		STATE_OPEN: 	(* Waiting for incomming connection *)
				m_SizeSockadr:=SIZEOF(m_AddressInfo);
				m_Socket:= SysSockAccept( m_ServerSocket, ADR(m_AddressInfo), ADR(m_SizeSockadr));
				diError:=State_open;
				IF m_Socket <> SOCKET_INVALID THEN
					xClientConnected:=TRUE;
					(*Set Push-Bit:new V1.5*)
					IF ADR(%MW0)=16#30000000  OR ADR(%MW0)=16#20000000 THEN (*841 or 881*)
						SysSockSetOption(
							diSocket:=m_Socket,
							diLevel:=6,
							diOption:=SOCKET_TCP_NODELAY,
							pOptionValue:=ADR(diOption),
							diOptionLength:=SIZEOF(diOption));
					ELSE
							;
					END_IF
					SysSockIoctl( m_Socket, SOCKET_FIONBIO, ADR(m_NoneBlocking));
					m_State:= STATE_RX;
					diError:=0;
				END_IF

		STATE_RX:
					m_BytesReceived:= SysSockRecv( m_Socket, ADR(m_ReceiveBuffer), SIZEOF(m_ReceiveBuffer), 0);
					CASE m_BytesReceived OF
					-1:(*no data available or error occured*)
						m_ConnectionWatchdog(IN:=TRUE , PT:=tServerTimeOut );
						IF m_connectionWatchdog.Q THEN
							m_State:= STATE_CLOSE;
							m_ConnectionWatchdog(IN:=FALSE);(*reset connection watchdog*)
							diError := 16#8009;
						END_IF
					0:(* socket was "gracefully closed"  *)
						m_State:= STATE_CLOSE;
						diError := 16#8003;
					ELSE
						(* Copy received data into receive buffer *)
						(********************************)
						FOR i:= 0 TO DINT_TO_INT(m_BytesReceived	)-1 DO
							aReceiveBuffer[diReceiveCount]:= m_ReceiveBuffer[i];
							diReceiveCount:=(diReceiveCount+1) MOD SIZEOF(aReceiveBuffer);
						END_FOR

						m_ConnectionWatchdog(IN:=FALSE);(*reset connection watchdog*)
					END_CASE

				(*send data*)
				IF xStartSend	 THEN
					m_State := STATE_TX;
				END_IF

	STATE_TX:	 (* send TCP-message *)
		m_diReturn := SysSockSend(diSocket := m_Socket,
								  pbyBuffer := ADR(ptSendData^[m_count]),(*geändert V1.4 bisher: [0] *)
								  diBufferSize := diSendCount-m_count,
								  diFlags :=m_Flags);
		CASE m_diReturn OF
		-1:	(* ERROR or data could not yet be send (V1.3 due to new FW11) *)
			m_ConnectionWatchdog(IN:=TRUE , PT:=tServerTimeOut );
			IF m_connectionWatchdog.Q THEN
				m_State:= STATE_CLOSE;
				m_ConnectionWatchdog(IN:=FALSE);(*reset connection watchdog*)
				diError := 16#8007;
			END_IF
		0: (* socket was "gracefully closed"  *)
			m_State := STATE_CLOSE;
			diError := 16#8003;
		ELSE (* succesful *)
			m_count:=m_count+m_diReturn;
			IF m_count>=diSendCount THEN
				diError := 16#0000;
				m_State := STATE_RX;
				m_count:=0;
				xStartSend:=FALSE;
			END_IF
			m_ConnectionWatchdog(IN:=FALSE);(*reset connection watchdog*)
		END_CASE


		STATE_CLOSE:	(* Close the server *)

		IF ADR(%MW0)=16#30000000  OR ADR(%MW0)=16#20000000 THEN (*841 or 881*)
			;
		ELSE
			IF m_Socket>=0 THEN
				SysSockShutdown(m_Socket, 0);;(*870*)
			END_IF
		END_IF
		IF m_Socket>=0 THEN
			SysSockClose( m_Socket);
		END_IF
		xClientConnected:= FALSE;
		m_State:= STATE_OPEN; (* Try to open the server again *)
		m_ConnectionWatchdog(IN:=FALSE);(*reset connection watchdog*)

		STATE_ERROR_TRAP: (* Error Read/Write socket  *)
			m_State:= STATE_ERROR_TRAP;

	ELSE  (* Bad FSM code trap  *)
			m_State:= STATE_ERROR_TRAP;
			diError:= 16#8008;
	END_CASE;
ELSE
	IF m_State <> STATE_INIT THEN
		IF ADR(%MW0)=16#30000000  OR ADR(%MW0)=16#20000000 THEN (*841 or 881*)
			;
		ELSE
			IF m_Socket>=0 THEN
				SysSockShutdown(m_Socket, 0);;(*870*)
			END_IF
		END_IF
		IF m_Socket>=0 THEN
			SysSockClose( m_Socket);
		END_IF
		IF ADR(%MW0)=16#30000000  OR ADR(%MW0)=16#20000000 THEN (*841 or 881*)
			;
		ELSE
			IF m_ServerSocket>=0 THEN
				SysSockShutdown(m_ServerSocket, 0);;(*870*)
			END_IF
		END_IF
		IF m_ServerSocket>=0 THEN
			SysSockClose( m_ServerSocket);
		END_IF
		xClientConnected:= FALSE;
		diError:= 0;
		m_State:= STATE_init; (* Try to open the server again *)
		m_ConnectionWatchdog(IN:=FALSE);(*reset connection watchdog*)
	END_IF
END_IF
END_FUNCTION_BLOCK

(* POU Utils Functions/HEXTORAW, ST *)
FUNCTION HEXTORAW : WORD
VAR_INPUT
	pString		: POINTER TO BYTE;
	StringLen	: WORD;
	pData		: POINTER TO BYTE;
END_VAR
VAR
	xl: WORD;
	xi: WORD;
	xr: BYTE;
END_VAR
xl:=0;
xi:=0;

WHILE xi<StringLen DO

	IF pString^>=97 AND pString^<=102 THEN
		xr := pString^ - 87;
	ELSIF pString^>=65 AND pString^<=70 THEN
		xr := pString^ - 55;
	ELSIF pString^>=48 AND pString^<=57 THEN
		xr := pString^ - 48;
	ELSE
		xr := 16;
	END_IF

	IF xr<16 THEN
		IF (xi AND 1)=0 THEN
			pData^ := xr * 16;
		ELSE
			pData^ := pData^ + xr;
			pData := pData + 1;
			xl := xl + 1;
		END_IF
	END_IF

	xi := xi + 1;
	pString := pString + 1;

END_WHILE

HEXTORAW:=xl;
END_FUNCTION

(* POU Utils Functions/RAWTOHEX, ST *)
FUNCTION RAWTOHEX : WORD
VAR_INPUT
	pData: POINTER TO BYTE;
	DataLen: WORD;
	pString: POINTER TO BYTE;
END_VAR
VAR
	xl: WORD;
END_VAR
xl:=0;

WHILE DataLen>0 DO

	pString^ := (pData^ / 16#10) + 48 + (((pData^ / 16#10)/10)*7);
	pString:=pString+1;
	pString^ := (pData^ AND 16#0F)  + 48 + (((pData^ AND 16#0F)/10)*7);
	pString:=pString+1;
	pData:=pData+1;
	DataLen:=DataLen-1;
	xl:=xl+2;

END_WHILE

(*pString^:=0;*)

RAWTOHEX:=xl;
END_FUNCTION

(* POU Utils Functions/SetDataTime, ST *)
FUNCTION SetDataTime : DT
VAR_INPUT
	year : INT;
	month : INT;
	day : INT;
	hour : INT;
	minute : INT;
	second : INT;
END_VAR

VAR
	count : INT;
END_VAR
(* Creazione variabiletipo DT per creare Orario da dare al PLC *)


IF month > 2 THEN
	count := (month - 1) * 30;
	IF month > 7 THEN count := count + SHR(month - 3,1); ELSE count := count + SHR(month - 4,1); END_IF;
	(* chech for leap year and add one day if true *)
	IF SHL(year,14) = 0 THEN count := count + 1; END_IF;
ELSE
	count := (month - 1) * 31;
END_IF;


SetDataTime := DWORD_TO_DT(DATE_TO_DWORD( DWORD_TO_DATE((INT_TO_DWORD(count + day - 1) + SHR(INT_TO_DWORD(year) * 1461 - 2878169, 2)) * 86400))
				+ INT_TO_DWORD(SECOND)
				+ INT_TO_DWORD(MINUTE) * 60
				+ INT_TO_DWORD(HOUR) * 3600);
END_FUNCTION

(* POU Utils/USRLED_Update, ST *)
PROGRAM USRLED_Update
VAR
	OldStatus: en_SYS_Status;

	aFS : ARRAY [0..24] OF FLASHING_SEQUENCE :=
		(Colour:=GREEN,  Frequency:=1,   Relation:=128, Duration:=t#0s,    NextIndex:=0),  (* 0 => RUNNING *)
		(Colour:=ORANGE, Frequency:=1,   Relation:=128, Duration:=t#0s,    NextIndex:=1),  (* 1 => INIT *)
		(Colour:=RED,    Frequency:=4,   Relation:=128, Duration:=t#0s,    NextIndex:=2),  (* 2 => ERROR *)
		(Colour:=RED,    Frequency:=10,  Relation:=128, Duration:=t#0s,    NextIndex:=3),  (* 3 => ALARM *)
		(Colour:=ORANGE, Frequency:=200, Relation:=16,  Duration:=t#100ms, NextIndex:=11), (* 10 *)
		(Colour:=ORANGE, Frequency:=200, Relation:=32,  Duration:=t#100ms, NextIndex:=12),
		(Colour:=ORANGE, Frequency:=200, Relation:=64,  Duration:=t#100ms, NextIndex:=13),
		(Colour:=ORANGE, Frequency:=200, Relation:=128, Duration:=t#100ms, NextIndex:=14),
		(Colour:=ORANGE, Frequency:=200, Relation:=192, Duration:=t#100ms, NextIndex:=15),
		(Colour:=ORANGE, Frequency:=200, Relation:=128, Duration:=t#100ms, NextIndex:=16),
		(Colour:=ORANGE, Frequency:=200, Relation:=64,  Duration:=t#100ms, NextIndex:=17),
		(Colour:=ORANGE, Frequency:=200, Relation:=32,  Duration:=t#100ms, NextIndex:=18),
		(Colour:=ORANGE, Frequency:=200, Relation:=16,  Duration:=t#100ms, NextIndex:=19),
		(Colour:=ORANGE, Frequency:=200, Relation:=8,   Duration:=t#100ms, NextIndex:=10),
		(Colour:=GREEN,  Frequency:=200, Relation:=16,  Duration:=t#100ms, NextIndex:=21), (* 20 *)
		(Colour:=GREEN,  Frequency:=200, Relation:=32,  Duration:=t#100ms, NextIndex:=22),
		(Colour:=GREEN,  Frequency:=200, Relation:=64,  Duration:=t#100ms, NextIndex:=23),
		(Colour:=GREEN,  Frequency:=200, Relation:=128, Duration:=t#100ms, NextIndex:=24),
		(Colour:=GREEN,  Frequency:=200, Relation:=192, Duration:=t#100ms, NextIndex:=25),
		(Colour:=GREEN,  Frequency:=200, Relation:=128, Duration:=t#100ms, NextIndex:=26),
		(Colour:=GREEN,  Frequency:=200, Relation:=64,  Duration:=t#100ms, NextIndex:=27),
		(Colour:=GREEN,  Frequency:=200, Relation:=32,  Duration:=t#100ms, NextIndex:=28),
		(Colour:=GREEN,  Frequency:=200, Relation:=16,  Duration:=t#100ms, NextIndex:=29),
		(Colour:=GREEN,  Frequency:=200, Relation:=8,   Duration:=t#100ms, NextIndex:=20);

	pFS : POINTER TO FLASHING_SEQUENCE;


END_VAR
IF Sys.Status <> OldStatus THEN

	OldStatus:=Sys.Status;

	CASE OldStatus OF

		S_STARTUP:
			pFS:=ADR(aFS);
			SET_FLASHING_SEQUENCE(EN:=TRUE, POINTER_TO_POINTER_TO_ARRAY:=ADR(pFS));
			SET_FLASHING_SEQUENCE_INDEX(EN:=TRUE, IMMEDIATE:=FALSE, INDEX:=1);
			START_FLASHING_SEQUENCE(EN:=TRUE);

		S_RUNNING:
			SET_FLASHING_SEQUENCE_INDEX(EN:=TRUE, IMMEDIATE:=TRUE, INDEX:=0);

	END_CASE

END_IF
END_PROGRAM

(* POU ConteggioGAS1, ST *)
PROGRAM ConteggioGAS1

VAR RETAIN
	Conteggio_GAS1: DINT;
END_VAR
(* Attenzione Portata GAS Caldaia n.3 SEVESO *)


Conteggio_GAS1:=Conteggio_GAS1+1;
END_PROGRAM
ACTION Offset:
(* Offset *)

IF ChangeGAS1 THEN
	Conteggio_GAS1:=OffsetGAS1;
	ChangeGAS1:=FALSE;
END_IF
END_ACTION

(* POU ConteggioGAS2, ST *)
PROGRAM ConteggioGAS2

VAR RETAIN
	Conteggio_GAS2: DINT;
END_VAR
(* Attenzione Portata GAS per Caldaia CAL02 e CAL03 *)

Conteggio_GAS2:=Conteggio_GAS2+1;
END_PROGRAM
ACTION Offset:
(* Offset *)

IF ChangeGAS2 THEN
	Conteggio_GAS2:=OffsetGAS2;
	ChangeGAS2:=FALSE;
END_IF
END_ACTION

(* POU Plant/SYS_Proc, ST *)
PROGRAM SYS_Proc
VAR
(*	fALARM_PB		:FLT_TAP;
	fALARM_TB		:FLT_TAP;
	fALARM_PM		:FLT_TAP; *)

(*	fGZB_ST			:FLT_TAP;  (* GATEWAY ZIGBEE *)*)
(*	fVPN_ST1		:FLT_TAP;  (* VPN CONNECT *)*)
	fVPN_ST2		:FLT_TAP;  (* VPN STATUS *)
(*	fKEY_CT_ST		:FLT_TAP;  (* DOOR1 *)*)
(*	fKEY_SCT_ST		:FLT_TAP;  (* DOOR2 *)*)
	fKEY_QE_ST		:FLT_TAP;  (* DOOR3 *)

END_VAR
(*************** ISPESL *****************)
(*
fALARM_PB(IN:=ALARM_PB);
IF fALARM_PB.EVH THEN
	LogEv(EL_AlarmStop,EO_PBV,1,1,'Over_Pressure_Alarm');
END_IF

fALARM_TB(IN:=ALARM_TB);
IF fALARM_TB.EVH THEN
	LogEv(EL_AlarmStop,EO_TBV,1,1,'Over_Temperature_Alarm');
END_IF

fALARM_PM(IN:=ALARM_PM);
IF fALARM_PM.EVH THEN
	LogEv(EL_AlarmStop,EO_PMV,1,1,'Under_Pressure_Alarm');
END_IF
*)
(****************************************)

(*### VPN Connection Check ###*)(*
fVPN_ST1(IN:=VPN_ST1);
IF fVPN_ST1.EVH THEN
	LogEv(EL_Log,EO_VPN,1,1,'CONNECT_ON');
END_IF
IF fVPN_ST1.EVL THEN
	LogEv(EL_Log,EO_VPN,1,2,'CONNECT_OFF');
END_IF*)

(*### VPN Status Check ###*)
fVPN_ST2(IN:=VPN_ST2);
IF fVPN_ST2.EVH THEN
	LogEv(EL_Log,EO_VPN,1,3,'STATUS_UP');
END_IF
IF fVPN_ST2.EVL THEN
	LogEv(EL_Wrn,EO_VPN,1,4,'STATUS_DOWN');
END_IF

(*### DOOR01 Status Check ###*)(*
fKEY_CT_ST(IN:=KEY_CT_ST);
IF fKEY_CT_ST.EVH THEN
	LogEv(EL_Log,EO_DOOR,1,2,'Centrale_termica_Close');
END_IF
IF fKEY_CT_ST.EVL THEN
	LogEv(EL_Wrn,EO_DOOR,1,1,'Centrale_termica_Open');
END_IF*)

(*### DOOR02 Status Check ###*)(*
fKEY_SCT_ST(IN:=KEY_SCT_ST);
IF fKEY_SCT_ST.EVH THEN
	LogEv(EL_Log,EO_DOOR,2,2,'Sottocentrale_termica_Close');
END_IF
IF fKEY_SCT_ST.EVL THEN
	LogEv(EL_Wrn,EO_DOOR,2,1,'Sottocentrale_termica_Open');
END_IF*)

(*### DOOR03 Status Check ###*)
fKEY_QE_ST(IN:=KEY_QE_ST);
IF fKEY_QE_ST.EVH THEN
	LogEv(EL_Log,EO_DOOR,3,2,'Quadro_Close');
END_IF
IF fKEY_QE_ST.EVL THEN
	LogEv(EL_Wrn,EO_DOOR,3,1,'Quadro_Open');
END_IF
END_PROGRAM

(* POU Utils Functions/AVERAGE_DINT, ST *)
FUNCTION_BLOCK AVERAGE_DINT
VAR_INPUT
	IN: 	DINT;
END_VAR
VAR_OUTPUT
	HI:		DINT;
	AVG:	DINT;
	LOW:	DINT;
	ERR:	BOOL;
END_VAR
VAR
	sum:	REAL;
	cnt:	WORD;
END_VAR
IF cnt>=65000 THEN
	ERR:=TRUE;
	Read();
	sum := sum - DINT_TO_REAL(AVG);
	cnt := cnt - 1;
END_IF

sum := sum + DINT_TO_REAL(IN);
cnt := cnt + 1;

IF IN<LOW THEN LOW:=IN; END_IF
IF IN>HI  THEN HI :=IN; END_IF
END_FUNCTION_BLOCK
ACTION Read:
AVG := REAL_TO_DINT(sum/cnt);
END_ACTION
ACTION Reset:
HI:=IN;
AVG:=IN;
LOW:=IN;
ERR:=FALSE;

sum:=DINT_TO_REAL(IN);
cnt:=1;
END_ACTION

(* POU Utils Functions/AVERAGE_INT, ST *)
FUNCTION_BLOCK AVERAGE_INT
VAR_INPUT
	IN: 	INT;
END_VAR
VAR_OUTPUT
	HI:		INT;
	AVG:	INT;
	LOW:	INT;
	ERR:	BOOL;
END_VAR
VAR
	sum:	DINT;
	cnt:	WORD;
END_VAR
IF cnt>=65000 THEN
	ERR:=TRUE;
	Read();
	sum := sum - AVG;
	cnt := cnt - 1;
END_IF

sum := sum + IN;
cnt := cnt + 1;

IF IN<LOW THEN LOW:=IN; END_IF
IF IN>HI  THEN HI :=IN; END_IF
END_FUNCTION_BLOCK
ACTION Read:
AVG := DINT_TO_INT(sum/cnt);
END_ACTION
ACTION Reset:
HI:=IN;
AVG:=IN;
LOW:=IN;
ERR:=FALSE;

sum:=IN;
cnt:=1;
END_ACTION

(* POU Utils Functions/AVERAGE_T, ST *)
FUNCTION_BLOCK AVERAGE_T
VAR_INPUT
	IN: 	INT;
END_VAR
VAR_OUTPUT
	HI:		INT;
	AVG:	INT;
	LOW:	INT;
	ERR:	BOOL;
END_VAR
VAR
	sum:	DINT;
	cnt:	WORD;
END_VAR
IF cnt>=65000 THEN
	ERR:=TRUE;
	Read();
	sum := sum - AVG;
	cnt := cnt + 1;
END_IF

sum := sum + IN;
cnt := cnt + 1;

IF IN<LOW THEN  LOW:=IN; END_IF
IF IN>HI  THEN HI :=IN; END_IF
END_FUNCTION_BLOCK
ACTION Read:
AVG := DINT_TO_INT(sum/cnt);
END_ACTION
ACTION Reset:
HI:=IN;
AVG:=IN;
LOW:=IN;
ERR:=FALSE;

sum:=IN;
cnt:=1;
END_ACTION

(* POU Utils Functions/COPY_32SWAP16, ST *)
FUNCTION COPY_32SWAP16:BOOL
VAR_INPUT
	pSourceAddress		:POINTER TO ARRAY[1..2] OF WORD;
	pDestinationAddress	:POINTER TO ARRAY[1..2] OF WORD;
END_VAR
VAR
END_VAR
pDestinationAddress^[1]:=pSourceAddress^[2];
pDestinationAddress^[2]:=pSourceAddress^[1];
END_FUNCTION

(* POU Utils/CSV_Log, ST *)
FUNCTION CSV_Log : BOOL
VAR_INPUT
END_VAR
VAR CONSTANT
	LogFileName:STRING:='S:\LOGS_ID3V3.CSV';
END_VAR
VAR
	s1 : STRING(180);
	hFile: 	DWORD;
END_VAR
(* Check file presence *)
hFile:=SysFileOpen(LogFileName,'r');
IF hFile=0 THEN
	(*** File not exist *** Create file and write header *)
	hFile:=SysFileOpen(LogFileName,'w');
	IF hFile<>0 THEN
		(* Write CSV header *)
		s1:='DATE-TIME;T-SA;T-S02;T-S03;T-S04;T-S05;T-S06;T-S07;';
		SysFileWrite(hFile, ADR(s1), LEN(s1));
		s1:='PORT01-Flow;PORT01-Cnt;GAS01-Cnt;GAS02-Cnt;';
		SysFileWrite(hFile, ADR(s1), LEN(s1));
		s1:='CTB250-Power;CTB250-KWH;CTB250-GWH';
		SysFileWrite(hFile, ADR(s1), LEN(s1));
		SysFileWrite(hFile, ADR(Logger_CRLF), LEN(Logger_CRLF));
	END_IF
ELSE
	(*** File exist *** Close file and reopen in append mode *)
	SysFileClose(hFile);
	hFile:=SysFileOpen(LogFileName,'a');
END_IF

(* Log to file *)
IF hFile<>0 THEN
	(* Date stamp *)
	s1:=REPLACE( Sys.Time_LogString , ' ' , 1 , 11 );
	SysFileWrite(hFile, ADR(s1), LEN(s1));
	(* Log data *)
	s1:=CONCAT(';', INT_TO_STRING(TT_S01) );
	s1:=CONCAT(s1 , ';' );
	s1:=CONCAT(s1 , INT_TO_STRING(TPV02.ValoreScalato) );
	s1:=CONCAT(s1 , ';' );
	s1:=CONCAT(s1 , INT_TO_STRING(TPV03.ValoreScalato) );
	s1:=CONCAT(s1 , ';' );
	s1:=CONCAT(s1 , INT_TO_STRING(TPV04.ValoreScalato) );
	s1:=CONCAT(s1 , ';' );
	s1:=CONCAT(s1 , INT_TO_STRING(TPV05.ValoreScalato) );
	s1:=CONCAT(s1 , ';' );
	s1:=CONCAT(s1 , INT_TO_STRING(TPV06.ValoreScalato) );
	s1:=CONCAT(s1 , ';' );
	s1:=CONCAT(s1 , INT_TO_STRING(TPV07.ValoreScalato) );
	SysFileWrite(hFile, ADR(s1), LEN(s1));
	s1:=CONCAT(';', DINT_TO_STRING(PORT01.ValoreScalato/1000) );
	s1:=CONCAT(s1 , ';' );
	s1:=CONCAT(s1 , DINT_TO_STRING(PortataTotalePORT01) );
	s1:=CONCAT(s1 , ';' );
	s1:=CONCAT(s1 , DINT_TO_STRING(ConteggioGAS1.Conteggio_GAS1) );
	s1:=CONCAT(s1 , ';' );
	s1:=CONCAT(s1 , DINT_TO_STRING(ConteggioGAS2.Conteggio_GAS2) );
(*	s1:=CONCAT(s1 , DINT_TO_STRING(PortataTotaleGAS01) );
	s1:=CONCAT(s1 , ';' );
	s1:=CONCAT(s1 , DINT_TO_STRING(PortataTotaleGAS02) );*)
	SysFileWrite(hFile, ADR(s1), LEN(s1));
	s1:=CONCAT(';', DINT_TO_STRING(REAL_TO_DINT(CTB250.POWER_KW)) );
	s1:=CONCAT(s1 , ';' );
	s1:=CONCAT(s1 , DWORD_TO_STRING(CTB250_ENERGY) );
	SysFileWrite(hFile, ADR(s1), LEN(s1));

	(* Add line CRLF and close *)
	SysFileWrite(hFile, ADR(Logger_CRLF), LEN(Logger_CRLF));
	SysFileClose(hFile);
END_IF
END_FUNCTION

(* POU Utils Functions/FLT_EVENT, ST *)
FUNCTION_BLOCK FLT_EVENT
VAR_INPUT
	IN		: BOOL;
	INITEV	: BOOL:=TRUE;
END_VAR
VAR_OUTPUT
	EVH		: BOOL;
	EVL		: BOOL;
END_VAR
VAR
	init	: BOOL:=FALSE;
	old		: BOOL;
END_VAR
EVH:=FALSE;
EVL:=FALSE;

IF NOT init THEN
	init:=TRUE;
	IF INITEV THEN
		old := NOT IN;
	ELSE
		old := IN;
	END_IF
END_IF

IF old<>IN THEN
	old:=IN;
	IF IN THEN EVH:=TRUE; ELSE EVL:=TRUE; END_IF
END_IF
END_FUNCTION_BLOCK

(* POU Utils Functions/FLT_TIME, ST *)
FUNCTION_BLOCK FLT_TIME
VAR_INPUT
	IN		: BOOL;
	TTAP	: TIME:=T#5s;
	INITEV	: BOOL:=TRUE;
END_VAR
VAR_OUTPUT
	OUT		: BOOL;
	EVH		: BOOL;
	EVL		: BOOL;
END_VAR
VAR
	init	: BOOL:=FALSE;
	timer	: TON;
END_VAR
EVH:=FALSE;
EVL:=FALSE;

IF NOT init THEN
	init := TRUE;
	IF INITEV THEN
		OUT  := NOT IN;
	ELSE
		OUT  := IN;
	END_IF
END_IF

IF OUT<>IN THEN
	timer(IN:=TRUE,PT:=TTAP);
	IF timer.Q THEN
		OUT:=IN;
		timer(IN:=FALSE);
		IF OUT THEN EVH:=TRUE; ELSE EVL:=TRUE; END_IF
	END_IF
ELSE
	timer(IN:=FALSE);
END_IF
END_FUNCTION_BLOCK

(* POU Utils Functions/LINEAR, ST *)
FUNCTION LINEAR : REAL (* Linear interpolation *)
VAR_INPUT
	X_In	: REAL;
	P1_X	: REAL;
	P1_Y	: REAL;
	P2_X	: REAL;
	P2_Y	: REAL;
END_VAR
VAR
END_VAR
LINEAR:=P1_Y+(((P2_Y-P1_Y)*(X_In-P1_X))/(P2_X-P1_X));
END_FUNCTION

(* POU Utils Functions/LINEAR_BAD, ST *)
FUNCTION LINEAR_BAD : INT (* Linear interpolation *)
VAR_INPUT
	PuntoMinX	: INT;
	PuntoMaxX	: INT;
	ValIn		: INT;
	PuntoMinY	: REAL;
	PuntoMaxY	: REAL;
	Decimali	: BYTE;
END_VAR
VAR
	Gain				: REAL;
	PuntoMinX_R			: REAL;
	PuntoMaxX_R			: REAL;
	Linearizzazione_R	: REAL;
END_VAR
PuntoMinX_R:=INT_TO_REAL(PuntoMinX);
PuntoMaxX_R:=INT_TO_REAL(PuntoMaxX);

Gain:=(PuntoMaxX_R-PuntoMinX_R)/(PuntoMaxY-PuntoMinY);	(* Calcolo in guadagno per la linarizzazione *)
Linearizzazione_R:=PuntoMinx+(Gain*(ValIn-PuntoMinY));	(* Ottengo il valore linearizzato *)

LINEAR_BAD:=REAL_TO_INT(Linearizzazione_R*(EXPT(10, Decimali)));  (* Ottengo intero con i decimai voluti *)
END_FUNCTION

(* POU TCP_Logger/LogTrig, ST *)
FUNCTION LogTrig : BOOL
VAR
	s1 : STRING(160);
	i  : BYTE;
END_VAR
(*---------------------------------------------------------------*)
	Logger_Head();
(*---------------------------------------------------------------*)

(* Insert TPVs *)
(*
s1:=CONCAT('&TPV=',INT_TO_STRING(TPV01.AVG));
(*TPV01.Mean_Reset(); *)
s1:=CONCAT(s1,';'); s1:=CONCAT(s1,INT_TO_STRING(TPV02.ValoreScalato));
s1:=CONCAT(s1,';'); s1:=CONCAT(s1,INT_TO_STRING(TPV03.ValoreScalato));
s1:=CONCAT(s1,';'); s1:=CONCAT(s1,INT_TO_STRING(TPV04.ValoreScalato));
s1:=CONCAT(s1,';'); s1:=CONCAT(s1,INT_TO_STRING(TPV05.ValoreScalato));
s1:=CONCAT(s1,';'); s1:=CONCAT(s1,INT_TO_STRING(TPV06.ValoreScalato));
s1:=CONCAT(s1,';'); s1:=CONCAT(s1,INT_TO_STRING(TPV07.ValoreScalato));
s1:=CONCAT(s1,';'); s1:=CONCAT(s1,INT_TO_STRING(TPV08.ValoreScalato));
s1:=CONCAT(s1,';'); s1:=CONCAT(s1,INT_TO_STRING(TPV09.ValoreScalato));

ADDSTRING(ADR(Logger.TData), ADR(s1), Logger.TLen);
*)

TPV01.AddLogData();
TPV02.AddLogData();
TPV03.AddLogData();
TPV04.AddLogData();
TPV05.AddLogData();
TPV06.AddLogData();
TPV07.AddLogData();
TPV08.AddLogData();
TPV09.AddLogData();

THER01.AddLogData();
THER02.AddLogData();
THER03.AddLogData();
THER04.AddLogData();

CIRD01.AddLogData();
CIRD02.AddLogData();

EV02.AddLogData();
EV03.AddLogData();

CAL02.AddLogData(CLIM:=CAL02_Clima);
CAL03.AddLogData(CLIM:=CAL03_Clima);

(* Insert contabilizers  *)

s1:=CONCAT('&PORT01=',DINT_TO_STRING(PORT01.ValoreScalato));
s1:=CONCAT(s1,';'); s1:=CONCAT(s1,DINT_TO_STRING(PortataTotalePORT01));
s1:=CONCAT(s1,';'); s1:=CONCAT(s1,BYTE_TO_STRING(PORT01.Status_Log));
ADDSTRING(ADR(Logger.TData), ADR(s1), Logger.TLen);


(*
s1:=CONCAT('&GAS01=',DINT_TO_STRING(PortataTotaleGAS01));
s1:=CONCAT(s1,';'); s1:=CONCAT(s1,BYTE_TO_STRING(GAS01.Status_Log));
ADDSTRING(ADR(Logger.TData), ADR(s1), Logger.TLen);

s1:=CONCAT('&GAS02=',DINT_TO_STRING(PortataTotaleGAS02));
s1:=CONCAT(s1,';'); s1:=CONCAT(s1,BYTE_TO_STRING(GAS02.Status_Log));
ADDSTRING(ADR(Logger.TData), ADR(s1), Logger.TLen);
*)

(* Registro il nuovo conteggio *)


s1:=CONCAT('&GAS01=',DINT_TO_STRING(ConteggioGAS1.Conteggio_GAS1));
s1:=CONCAT(s1,';'); s1:=CONCAT(s1,BYTE_TO_STRING(GAS01.Status_Log));
ADDSTRING(ADR(Logger.TData), ADR(s1), Logger.TLen);

s1:=CONCAT('&GAS02=',DINT_TO_STRING(ConteggioGAS2.Conteggio_GAS2));
s1:=CONCAT(s1,';'); s1:=CONCAT(s1,BYTE_TO_STRING(GAS02.Status_Log));
ADDSTRING(ADR(Logger.TData), ADR(s1), Logger.TLen);


(*CTBSCAN01.AddLogData( MBUS:=MBUS01 ); ==> TOO BIG! *)
CTB250.AddLogData( ENERGY_WH:=CTB250_ENERGY_WH,	ENERGY:=CTB250_ENERGY );

SCA_Proc.AddLogData();

(*---------------------------------------------------------------*)
	Logger_Send();
(*---------------------------------------------------------------*)
END_FUNCTION

(* POU Utils Functions/MEMCLR, ST *)
FUNCTION MEMCLR:BOOL
VAR_INPUT
	pDestinationAddress:POINTER TO ARRAY[1..2] OF BYTE;
	BytesToClear:WORD;
END_VAR
VAR
END_VAR
WHILE (BytesToClear > 0) DO
	pDestinationAddress^[1]:=0;
	pDestinationAddress:=ADR(pDestinationAddress^[2]); (* increment destination *)
	BytesToClear:=BytesToClear -1; (* decrement number of bytes to copy *)
END_WHILE
END_FUNCTION

(* POU Plant_Objects/obj_CAL_01, ST *)
FUNCTION_BLOCK obj_CAL_01
(* === CALDAIA generica con comando digitale, Set point analogico feedback potenza e stato caldaia  ===
   VERSIONE 01 REALIZZATA DA MORENO E TESTA SU IMPIANTO SAN FELICE ID 003 CLV
	Caldaia controllata con: 	- uscita analogica
								- comando on/off. 
								- Reset Blocco Bruciatore
	
	come feedback si sapetta: 	- riferimento analogico per potenza
								- Stato Presenza fiamma per segnalazione Caldaia accesa
								- Stato Blocco Brucitaore
*)
VAR_INPUT

	ID				: BYTE;			(* Impostazione *)
	LimiteMAXSetPoint: INT;			(* Da Settare : limite massimo da assegnare al riferimento analogico onde evitare di mal comndare la caldaia *)
	LimiteMinSetPoint: INT;			(* Da Settare : limite massimo da assegnare al riferimento analogico onde evitare di mal comndare la caldaia *)

	SetPointManuale: INT; 			(* SetPoint forazato in manuale serve per escludere la curva climatica locale *)
	AbilitaSetPointManuale : BOOL ; (* Abilita il funzionamento col set point Manaule Escludendo la curva cliamtica *)

	Run				: BOOL;			(* Controllo/ comando esterno generalmente da Crono *)


(* ingressi fisici analogici *)

	AI_Potenza		:INT;			(* Riferimento della potenza erogata dalla Caldaia *)

(* ingressi fisici digitali *)

	CAL_ST : BOOL;					(* Stato della Caldia Accesa Spenta - Presenza Fiamma *)
	ALARM_CAL:BOOL;					(* Caldaia in BLocco  *)
	PresenzaFiamma:BOOL;			(* Segnalazione Presenza Fiamma *)


	CmdCALAuto_MAN: BOOL;			(* Modalaita di Funzionamento Caldaia : 0 Automatico. 1 Manuale Solitamnete Selettore a bordo Caldaia *)

	TCP_ResetCAL:BOOL;				(* Comando Reset Caldaia da Remoto via FTP *)
	Rearm:BOOL;						(* Comando Reset Caldaia da locale pulsante WebVisu *)

END_VAR
VAR_IN_OUT
	CLIM		  : typ_Clima;
END_VAR
VAR_OUTPUT
	Curve_Temp		: INT;
	AO_SetPoint		:INT;

	CAL_EN			:BOOL;
	DO_RIARMO		:BOOL;

	(* Status *)
	Status_Log	: BYTE;
	Status_Vis 	: DWORD;
END_VAR
VAR
	InitOK		: BOOL;

	Alarm: BOOL;
	Warning:BOOL;
	Warning2: BOOL;

	Curve 		: CHARCURVE;
	Curve_Err 	: BYTE;


	(* Timer manage switch on/off delay *)
	Delay		: 	TONOF;


	Potenza:INT;
	SetPoint:INT;

	fSTATO_CAL: FLT_TAP;
	fALARM_CAL: FLT_TAP;
	fCALAuto_MAN: FLT_TAP;



	TP_RIARMO: TP:=(PT:=t#5s);



	MAXTentativi: BYTE;
	Trig_TP_RIARMO: R_TRIG;




END_VAR

VAR_INPUT RETAIN

	(* Timings *)
	OnDelay		:	TIME;	(* Switch on delay *)
	OffDelay	:	TIME;	(* Switch off delay *)


END_VAR
(* Check initialization *)
(*IF NOT InitOK THEN Init(); END_IF*)

(* Recupero della curva cliamtica *)

IF NOT CLIM.InitOK THEN Clima_Default(); END_IF;
(* Calculate Setpoint *)
Curve(	IN:= T_AMB,	N:= 5, P:= CLIM.Points,
		OUT=> Curve_Temp, ERR=> Curve_Err );
IF Curve_Err>0  THEN
	IF NOT Warning THEN
		Warning:=TRUE;
		LogEv(EL_Wrn,EO_CAL,ID,2,'Climatic_Error');
	END_IF
ELSE
	Warning:=FALSE;
END_IF


(* Scelta del set point della cladaia o vien preso dalla curva cliamtica o da un riferimento esterno *)
IF AbilitaSetPointManuale THEN
	SetPoint:=(SetPointManuale + OffsetSetPointManuale);
ELSE
	SetPoint:=Curve_Temp*10;
END_IF


(* Linearizzazione segnali analogici *)

(* calcolao il valore delset point da passare alla scheda di uscita  analogica *)
SetPoint:=LIMIT(LimiteMinSetPoint,SetPoint,LimiteMAXSetPoint);
AO_SetPoint:=LINEAR_BAD(0, 32767, SetPoint, 0,1500 , 0);

(* trovo Valore della potenza della Caldaia *)
Potenza:=LINEAR_BAD(0, 100, AI_Potenza, 6553, 32767, 0);
Potenza:=LIMIT(0,Potenza,100);




(* Comando fisico alla caldaia Solito Ton e TOFF *)
IF OffDelay<t#1s THEN OffDelay:=t#1s;END_IF;
IF OnDelay<t#1m THEN OffDelay:=t#1m;END_IF;

Delay(IN:=RUN,PT_OF:=OffDelay,PT_ON:=OnDelay + WORD_TO_TIME(1000*ID));    (* Ritardo all'accensione e allo Spegnimento *)

(* Controllo On/Off Caldaia *)
IF Delay.OUT AND (NOT Alarm) AND NOT CmdCALAuto_MAN THEN
	CAL_EN:=TRUE;
 ELSE
	CAL_EN:=FALSE;
END_IF


(** Riarmo Reset Caldaia tolgo tensione per 5 secondi alla caldaia ***)

TP_RIARMO(IN:=Rearm OR TCP_ResetCAL AND ALARM_CAL );
DO_RIARMO:=TP_RIARMO.Q;
Rearm:=FALSE;
TCP_ResetCAL:=FALSE;

Trig_TP_RIARMO(CLK:=TP_RIARMO.Q);
IF Trig_TP_RIARMO.Q THEN MAXTentativi:=MAXTentativi+1;END_IF
IF MAXTentativi >5 THEN
	LogEv(EL_Alarm,EO_CAL,ID,14,'Reset_Caldaia_non_riuscito');
	MAXTentativi:=0;
END_IF

(* Stato CALDAIA *)
fALARM_CAL(IN:=ALARM_CAL);
IF fALARM_CAL.EVH THEN
	LogEv(EL_Alarm,EO_CAL,ID,5,'Caldaia_In_Blocco');
	Alarm:=TRUE;
END_IF
IF fALARM_CAL.EVL THEN
	LogEv(EL_Alarm,EO_CAL,ID,6,'CALDAIA_Sbloccata');
	MAXTentativi:=0;
	Alarm:=FALSE;
END_IF

(* Stato CALDAIA CALDAIA in Mauale  *)
fCALAuto_MAN(IN:=CmdCALAuto_MAN);
IF fCALAuto_MAN.EVH THEN
	LogEv(EL_wrn,EO_CAL,ID,12,'Caldaia_In_Manuale');
	Warning2:=TRUE;
END_IF
IF fCALAuto_MAN.EVL THEN
	LogEv(EL_Log,EO_CAL,ID,13,'CALDAIA_in_Automatico');
	Warning2:=FALSE;
END_IF


(* Stato CALDAIA *)
fSTATO_CAL(IN:=CAL_ST);
IF fSTATO_CAL.EVH THEN
	LogEv(EL_Log,EO_CAL,ID,10,'Caldaia_RUN_Presenza_Fiamma');
	MAXTentativi:=0;
END_IF
IF fSTATO_CAL.EVL THEN
	LogEv(EL_Log,EO_CAL,ID,11,'CALDAIA_STOP_Assenza_Fiamma');
END_IF



(* Seganalzione stato Caldaia *)
  IF Alarm THEN
		Status_Log:=2; Status_Vis:=16#2020F0;
		AO_SetPoint:=0;
	ELSIF Warning OR Warning2 THEN
			Status_Log:=1; Status_Vis:=16#20F0F0;
    ELSE
		Status_Log:=0;
		Status_Vis:=16#006000;
END_IF
END_FUNCTION_BLOCK
ACTION AddLogData:
Logger.s1:=INSERT('&CAL=',BYTE_TO_STRING(ID),4);
IF ID<10 THEN Logger.s1:=INSERT(Logger.s1,'0',4); END_IF

Logger.s1:=CONCAT(Logger.s1,INT_TO_STRING(SetPoint));
Logger.s1:=CONCAT(Logger.s1,';');
Logger.s1:=CONCAT(Logger.s1,SEL(Run,'0','100'));
Logger.s1:=CONCAT(Logger.s1,';');

Logger.s1:=CONCAT(Logger.s1,WORD_TO_STRING(Status_Log));

Logger.s1:=CONCAT(Logger.s1,';');
Logger.s1:=CONCAT(Logger.s1,INT_TO_STRING(OffsetSetPointManuale));			(* non pesente in quanto non c'è lo scambiatore *)
Logger.s1:=CONCAT(Logger.s1,';');
Logger.s1:=CONCAT(Logger.s1,INT_TO_STRING(Potenza)); 						(* Potenza Caldaia *)
Logger.s1:=CONCAT(Logger.s1,';');
Logger.s1:=CONCAT(Logger.s1,INT_TO_STRING(BOOL_TO_INT(PresenzaFiamma))); 				(* Presenza Fiamma *)
Logger.s1:=CONCAT(Logger.s1,';');
Logger.s1:=CONCAT(Logger.s1,INT_TO_STRING(0)); 								(* non recuperabile Temp. Mandata da Caldaia*)
Logger.s1:=CONCAT(Logger.s1,';');
Logger.s1:=CONCAT(Logger.s1,'3');	 											(* Temp. Tipo Caldaia Sempre in questo punto
																				0 = > Albino
																				1 = > Caldaia con Protocollo LON
																				2 = > comandi digitali senza set point 
																				3 = > comandi digitali con set point *)
Logger.s1:=CONCAT(Logger.s1,';');
Logger.s1:=CONCAT(Logger.s1,INT_TO_STRING(BOOL_TO_INT(CmdCALAuto_MAN)));	 					(* 0 caldia in Automatico : 1= Caldaia in Manuale *)



ADDSTRING(ADR(Logger.TData), ADR(Logger.s1), Logger.TLen);
END_ACTION
ACTION Clima_Default:
IF CLIM.Points[0].X=0 THEN
CLIM.Points[0].X:=-100; CLIM.Points[0].Y:=800;
CLIM.Points[1].X:=0 ; CLIM.Points[1].Y:=750;
CLIM.Points[2].X:= 100;  CLIM.Points[2].Y:=700;
CLIM.Points[3].X:= 150; CLIM.Points[3].Y:=650;
CLIM.Points[4].X:= 200; CLIM.Points[4].Y:=400;
END_IF
CLIM.InitOK:=TRUE;
LogEv(EL_Wrn,EO_CAL,ID,1,'Climatic_default');
END_ACTION
ACTION Init:
(* End initialization *)
InitOK:=TRUE;
END_ACTION

(* POU Utils Functions/TONOF, ST *)
FUNCTION_BLOCK TONOF
VAR_INPUT
	IN		: BOOL;
	PT_ON	: TIME; (* time to pass, before OUT is set *)
	PT_OF	: TIME; (* time to pass, before OUT is reset *)
END_VAR
VAR_OUTPUT
	OUT		: BOOL;
END_VAR
VAR
	timer	: TON;
END_VAR
IF IN<>OUT THEN
	timer(IN:=TRUE,PT:=SEL(IN,PT_OF,PT_ON));
	IF timer.Q THEN OUT:=IN; END_IF
ELSE
	timer(IN:=FALSE);
END_IF
END_FUNCTION_BLOCK

(* POU Plant_Objects/obj_CIRD_01, ST *)
FUNCTION_BLOCK obj_CIRD_01
(* === CIRCOLATORE GEMELLARE STANDARD ===
   VERSIONE 01 REALIZZATA DA MORENO E TESTA SU IMPIANTO SAN FELICE ID 003 CLV
*)

VAR_INPUT
	(* Settings *)
	ID				: BYTE;

	(* Forzature da FTP *)
	CIR_RUN_REQ		: BOOL; (* Richiesta di avvio Circolatore  - Vince sullo stato del ciclo *)
	CIR_STOP_REQ	: BOOL; (* Richiesta di Stop Circolatore - Vince sullo stato del ciclo *)

	(* Ingressi Fisici  *)
	PumpA_AL		: BOOL; (* Allarme Pump A - Salvamotore Intervenuto *)
	PumpB_AL		: BOOL; (* Allarme Pump B - Salvamotore Intervenuto *)
	PumpA_ST		: BOOL; (* Stato Pump A - Generalmente Stato del Contattore *)
	PumpB_ST		: BOOL; (* Stato Pump B - Generalmente Stato del Contattore *)
	PumpA_AUTO		: BOOL; (* Pump A in 1=Automatico o 0=Manuale *)
	PumpB_AUTO		: BOOL; (* Pump B in 1=Automatico o 0=Manuale *)

	(* Controls *)
	OnOff			: BOOL;		(* On/Off from chrono *)
	Mode			: BYTE;   	(*			0 = Circolatore A ON e Ciroclatore B ON
											1 = Circolatori  in Automatico con con scambia a tempo e a causa di Allarme
											2 = Circolatore A ON e Ciroclatore B in Scorta 
											3 = Circolatore B ON e Ciroclatore A in Scorta 
											
											 *)

(* Working mode: 0-Both pumps works simultaneously, 1-Alternate every 24h, 2-Master/Backup *)

	InitOK			: BOOL;


END_VAR
VAR_OUTPUT
	PumpA_En		: BOOL;			(* uscita del ciclo *)
	PumpB_En		: BOOL;			(* uscita del ciclo *)

	Ctrl_Run		:	BOOL;		(* ritrasmissione dello stato OnOff  *)
	Run				:	BOOL;		(* Real status *)

	Status_Log		: WORD;
	Status_Vis		: DWORD;
END_VAR
VAR
	Pump_En		:	ARRAY [1..2] OF BOOL;

	ChangeTmr	: 	TON := (PT:=T#24h);				(* Timer that counts change time when in alternate mode *)
	ActivePump	: 	BYTE := 1;						(* Actual active pump *)
	NewActivePump	: BYTE := 1;

(*

	CIR_AUTO	: BOOL; (* Auto/Manual input signal *)

	(* Filters *)
	fPump_ST	: 	ARRAY [1..2] OF FLT_TIME := (INITEV:=FALSE);
	fPump_En	:	ARRAY [1..2] OF FLT_EVENT;
	fCIR_AUTO	:	ARRAY [1..2] OF FLT_TAP;
	fStatus		:	FLT_EVENT;
	fStatusFault:	BOOL;


	(* Alarm and Warning counters *)
	AlarmCtr	:	BYTE;
	WarningCtr	:	BYTE;


	(* Variables for status reconstruction *)
	aTprobe		:	ARRAY [1..SampleNr] OF INT;
	sample		:	BYTE;
	Tmean		:	INT;
	sum			:	INT;
	i			:	BYTE;
	moreno: BOOL; *)

	(* Filers on alarms and faults *)
	FLT_TAP_AllarmeHW_C1		: FLT_TAP := (INITEV:=FALSE);
	FLT_TAP_AllarmeHW_C2		: FLT_TAP := (INITEV:=FALSE);
	fPump_ST	: 	ARRAY [1..2] OF FLT_TIME := (INITEV:=FALSE);
	fCIR_AUTO	:	ARRAY [1..2] OF FLT_TAP;
	fBackup		:	FLT_EVENT := (INITEV:=FALSE);


	(* Timer manage switch on/off delay *)
	Delay		: 	TONOF;

	AllarmeHW_C1: BOOL;
	AllarmeHW_C2: BOOL;
	AllarmeHW2_C1: BOOL;
	AllarmeHW2_C2: BOOL;

	WarningP1_inMan:BOOL;
	WarningP2_inMan:BOOL;


	ScambioPompa: BOOL;
	PausaScambio: TP; (* Timer per implementare un piccolo ritardo fra lo scambio delle pompe *)

	BitAppoggioPump_2: BOOL; (* Bit Utili per la commutazione della pompa in automatico *)
	BitAppoggioPump_1: BOOL;


END_VAR
VAR_INPUT RETAIN
	(* Timings *)
	OnDelay		:	TIME;	(* Switch on delay *)
	OffDelay	:	TIME;	(* Switch off delay *)
END_VAR
Init();

PumpManager();

(* Check alarms and warnings *)
CheckFault();

IF ( AllarmeHW_C1 AND AllarmeHW_C2) OR  ( AllarmeHW2_C1 AND AllarmeHW2_C2) THEN
	Status_Log := 2;
	Status_Vis := COLOR_RED;
ELSIF WarningP1_inMan OR WarningP2_inMan  OR AllarmeHW_C1 OR AllarmeHW_C2 OR  AllarmeHW2_C1 OR AllarmeHW2_C2 THEN
	Status_Log := 1;
	Status_Vis := COLOR_YELLOW;
ELSE
	Status_Log := 0;
	Status_Vis := COLOR_GREEN;
END_IF
END_FUNCTION_BLOCK
ACTION AddLogData:
Logger.s1:=INSERT('&CIRD=',BYTE_TO_STRING(ID),5);
IF ID<10 THEN Logger.s1:=INSERT(Logger.s1,'0',5); END_IF

Logger.s1:=CONCAT(Logger.s1,WORD_TO_STRING(Mode));			Logger.s1:=CONCAT(Logger.s1,';');

Logger.s1:=CONCAT(Logger.s1,SEL(Pump_En[1],'0','100'));		Logger.s1:=CONCAT(Logger.s1,';');
Logger.s1:=CONCAT(Logger.s1,SEL(Pump_En[2],'0','100'));		Logger.s1:=CONCAT(Logger.s1,';');

Logger.s1:=CONCAT(Logger.s1,WORD_TO_STRING(Status_Log));
Logger.s1:=CONCAT(Logger.s1,';');
Logger.s1:=CONCAT(Logger.s1,SEL(CIR_RUN_REQ,'0','100'));
Logger.s1:=CONCAT(Logger.s1,';');
Logger.s1:=CONCAT(Logger.s1,SEL(CIR_STOP_REQ,'0','100'));




ADDSTRING(ADR(Logger.TData), ADR(Logger.s1), Logger.TLen);
END_ACTION
ACTION CheckFault:
(*** ALARMS ***)

(**** CIROCOLATORE 1 ****)
(* Allarme Hardware da ingresso PLC *)
FLT_TAP_AllarmeHW_C1(IN:=PumpA_AL);

IF FLT_TAP_AllarmeHW_C1.EVH THEN
	LogEv(EL_Alarm,EO_CIRD,ID,3,'Scatto_Termico_PompaA');
	AllarmeHW_C1 := TRUE;    (* Indice stato Allarme *)
END_IF

IF FLT_TAP_AllarmeHW_C1.EVL THEN
	LogEv(EL_Log,EO_CIRD,ID,4,'Termico_Riarmato_PompaA');
	AllarmeHW_C1 := FALSE;
END_IF

(**** CIRCOLATORE 2 ****)
(* Allarme Hardware da ingresso PLC *)
FLT_TAP_AllarmeHW_C2(IN:=PumpB_AL);

IF FLT_TAP_AllarmeHW_C2.EVH THEN
	LogEv(EL_Alarm,EO_CIRD,ID,3,'Scatto_Termico_PompaB');
	AllarmeHW_C2 := TRUE;   (* Indice stato Allarme *)
END_IF

IF FLT_TAP_AllarmeHW_C2.EVL THEN
	LogEv(EL_Log,EO_CIRD,ID,4,'Termico_Riarmato_PompaB');
	AllarmeHW_C2 := FALSE; ;
END_IF


(* Verify if in Auto or Manual mode *)
fCIR_AUTO[1](IN:=PumpA_AUTO);
fCIR_AUTO[2](IN:=PumpB_AUTO);

(*** Pump A ***)
IF fCIR_AUTO[1].EVH THEN
	LogEv(EL_Log,EO_CIRD,ID,8,'PompaA_in_AUTOMATIC_MODE');
	WarningP1_inMan := FALSE;
END_IF

(* Manual -> Keep switched on *)
IF fCIR_AUTO[1].EVL THEN
	LogEv(EL_Wrn,EO_CIRD,ID,7,'PumpaA_in_MANUAL_MODE');
	WarningP1_inMan := TRUE;
END_IF

(*** Pump B ***)
IF fCIR_AUTO[2].EVH THEN
	LogEv(EL_Log,EO_CIRD,ID,8,'PompaB_in_AUTOMATIC_MODE');
	WarningP2_inMan:=FALSE;
END_IF

(* Manual -> Keep switched on *)
IF fCIR_AUTO[2].EVL THEN
	LogEv(EL_Wrn,EO_CIRD,ID,7,'PumpaB_in_MANUAL_MODE');
	WarningP2_inMan:=TRUE;
END_IF


(* nella condizione di pompe in scorta (Mode>0) segnalo l'interventod della pompa in scorta*)
fBackup(IN:=(Mode>0 AND AllarmeHW_C2 OR AllarmeHW_C1));
IF fBackup.EVH THEN
	LogEv(EL_Wrn,EO_CIRD,ID,16,'Pompa_Scorta_Avviata');
END_IF



(* segnalazione discrepanza fra stato comando e stato teleruttore *)
fPump_ST[1](IN:=(PumpA_ST<>PumpA_EN));
	IF fPump_ST[1].EVH THEN
		IF PumpA_AUTO THEN
			LogEv	(SEL(PumpA_ST,EL_Alarm,EL_Wrn),
					EO_CIRD,
					ID,
					SEL(PumpA_ST,5,6),
					SEL(PumpA_ST ,'StatoTeleruttoreA_OFF','StatoTeleruttoreA_ON')
					);
			AllarmeHW2_C1 := (PumpA_ST);    (* Se il teleuttore non si è chiuso segnalo l'allarme *)
		ELSE
			LogEv(	EL_Wrn,
					EO_CIRD,
					ID,
					SEL(PumpA_ST,1,2),
					SEL(PumpA_ST ,'ComandoManualeA_OFF','ComandoManualeA_ON')
				);
		END_IF
	END_IF
	IF fPump_ST[1].EVL AND AllarmeHW2_C1  AND PumpB_EN=PumpA_ST THEN
		AllarmeHW2_C1:=FALSE;
	END_IF;


fPump_ST[2](IN:=(PumpB_ST<>PumpB_EN));

	IF fPump_ST[2].EVH THEN
		IF PumpB_AUTO THEN
			LogEv(SEL(PumpB_ST,EL_Alarm,EL_Wrn),EO_CIRD,ID,SEL(PumpB_ST,5,6),SEL(PumpB_ST,'StatoTeleruttoreB_OFF','StatoTeleruttoreB_ON'));
			AllarmeHW2_C2 := (PumpB_ST);    (* Se il teleuttore non si è chiuso segnalo l'allarme *)
		ELSE
			LogEv(EL_Wrn,EO_CIRD,ID,SEL(PumpB_ST,1,2),SEL(PumpB_ST,'ComandoManualeB_OFF','ComandoManualeB_ON'));
		END_IF
	END_IF

	IF fPump_ST[2].EVL AND AllarmeHW2_C2  AND PumpB_EN=PumpB_ST THEN
		AllarmeHW2_C2:=FALSE;
	END_IF;
END_ACTION
ACTION Init:
IF NOT InitOK THEN

	Pump_En[1] := FALSE;
	Pump_En[2] := FALSE;

	InitOK := TRUE;

END_IF
END_ACTION
ACTION PumpManager:
(* Verify if OnOff is changed *)
Ctrl_Run := OnOff;

(* Check switch on or switch off delay *)

IF OffDelay<t#5ms THEN OffDelay:=t#10ms;END_IF;
Delay(IN:=Ctrl_Run,PT_OF:=OffDelay,PT_ON:=OnDelay + WORD_TO_TIME(1000*ID));    (* Ritardo all'accensione e allo Spegnimento *)

(* Gestione delle pompe in funzione di quanto richiesto  	0 = Circolatore A ON e Ciroclatore B ON in Simultanea
															1 = Circolatori  in Automatico con con scambia a tempo e a causa di Allarme 
															2 = Circolatore A ON e Ciroclatore B in Scorta
															3 = Circolatore A in Scorta e Ciroclatore B ON *)


CASE Mode OF

		0:	(*0 = Circolatore A ON e Ciroclatore B ON in funzionamento Simultaneo *)
			IF PumpA_AUTO THEN (* Con Pompa gestita in Automatico dal PLC *)
				IF CIR_STOP_REQ THEN Pump_En[1] := FALSE;    (* solito gioco per forzare il Funzionemento della pompa da remoto il comando *)
				ELSIF CIR_RUN_REQ THEN Pump_En[1] := TRUE;
				ELSE Pump_En[1] := Delay.OUT;
				END_IF
			END_IF

			IF PumpB_AUTO THEN
				IF CIR_STOP_REQ THEN Pump_En[2] := FALSE;
				ELSIF CIR_RUN_REQ THEN Pump_En[2] := TRUE;
				ELSE Pump_En[2] := Delay.OUT;
				END_IF
			END_IF


		1:	(*1 = Circolatori  in Automatico con con scambia a tempo e a causa di Allarme *)

			(* Tempo ciclo per il lo scambio Automatico delle Pompe *)
				ChangeTmr(IN:=NOT ChangeTmr.Q);

				IF ChangeTmr.Q  THEN
					ScambioPompa:=NOT ScambioPompa;
				 (*	ChangeTmr.PT := T#24h; *)
				END_IF

			(* Questo tempo serve per avere un ritardo fisico sulla commutazione *)
				PausaScambio(IN:=ChangeTmr.Q OR AllarmeHW_C1 OR AllarmeHW_C2 OR AllarmeHW2_C1 OR AllarmeHW2_C2, PT:=t#3s , Q=> , ET=> );

							(* Il bit va a true quando *)
				BitAppoggioPump_1:=(ScambioPompa							(* Ho la commutazione a tempo *)
									OR( NOT AllarmeHW_C1 AND AllarmeHW_C2 )	(* Se non è presente l'allarme e non è comparso quella dell'alatra pompa *)
									OR( NOT AllarmeHW2_C1 AND AllarmeHW2_C2 ))(* Se è presente l'allarme di stato contattore *)
									AND NOT PausaScambio.Q						(* Finestra della pausa fra lo scambio delle pompe *)
									;
				BitAppoggioPump_2:=( NOT ScambioPompa							(* Ho la commutazione a tempo *)
									OR( NOT AllarmeHW_C2 AND AllarmeHW_C1 )	(* Se non è presente l'allarme e non è comparso quella dell'alatra pompa *)
									OR( NOT AllarmeHW2_C2 AND AllarmeHW2_C1))(* Se è presente l'allarme di stato contattore *)
									AND NOT PausaScambio.Q;					(* Finestra della pausa fra lo scambio delle pompe *)


			IF PumpA_AUTO THEN (* Con Pompa gestita in Automatico dal PLC *)
				IF CIR_STOP_REQ THEN
						 Pump_En[1] := FALSE;    (* solito gioco per forzare il Funzionemento della pompa da remoto il comando *)
				ELSIF CIR_RUN_REQ THEN
						Pump_En[1] := TRUE;
				ELSE
					Pump_En[1]:=Delay.OUT AND BitAppoggioPump_1;
				END_IF
			END_IF

			IF PumpB_AUTO THEN
				IF CIR_STOP_REQ THEN
						 Pump_En[2] := FALSE;
				ELSIF CIR_RUN_REQ THEN
						Pump_En[2] := TRUE ;
				ELSE
					Pump_En[2]:=Delay.OUT AND BitAppoggioPump_2;
				END_IF
			END_IF

		2:	(*2 = Circolatore A ON e Ciroclatore B in Scorta *)


			(* Questo tempo serve per avere un ritardo fisico sulla commutazione *)
				PausaScambio(IN:= AllarmeHW_C1 OR AllarmeHW2_C1 , PT:=t#3s , Q=> , ET=> );

																			(* Il bit va a true quando *)
				BitAppoggioPump_1:=(NOT AllarmeHW_C1 )						(* Se non è presente l'allarme Salvamotore *)
									AND NOT AllarmeHW2_C1					(* Se non è presente l'allarme Contattore *)
									AND NOT PausaScambio.Q;					(* Finestra della pausa fra lo scambio delle pompe *)

				BitAppoggioPump_2:= NOT BitAppoggioPump_1					(* se la pompa 1 ha dei problemi *)
									AND NOT AllarmeHW_C2					(* Se non è presente l'allarme Salvamotore *)
									AND NOT AllarmeHW2_C2					(* Se non è presente l'allarme Contattore *)
									AND NOT PausaScambio.Q;					(* Finestra della pausa fra lo scambio delle pompe *)


			IF PumpA_AUTO THEN (* Con Pompa gestita in Automatico dal PLC *)
				IF CIR_STOP_REQ THEN
						 Pump_En[1] := FALSE;    (* solito gioco per forzare il Funzionemento della pompa da remoto il comando *)
				ELSIF CIR_RUN_REQ THEN
						Pump_En[1] := TRUE AND ScambioPompa;
				ELSE
					Pump_En[1]:=Delay.OUT AND BitAppoggioPump_1;
				END_IF
			END_IF

			IF PumpB_AUTO THEN
				IF CIR_STOP_REQ THEN
						 Pump_En[2] := FALSE;
				ELSIF CIR_RUN_REQ THEN
						Pump_En[2] := TRUE AND NOT ScambioPompa;
				ELSE
					Pump_En[2]:=Delay.OUT AND BitAppoggioPump_2;
				END_IF
			END_IF



		3:	(*3 = Circolatore A in Scorta e Ciroclatore B ON *)


			(* Questo tempo serve per avere un ritardo fisico sulla commutazione *)
				PausaScambio(IN:= AllarmeHW_C2 , PT:=t#3s , Q=> , ET=> );

																			(* Il bit va a true quando *)


				BitAppoggioPump_2:=(NOT AllarmeHW_C2 )						(* Se non è presente l'allarme Salvamotore *)
									AND NOT AllarmeHW2_C2					(* Se non è presente l'allarme Contattore *)
									AND NOT PausaScambio.Q;					(* Finestra della pausa fra lo scambio delle pompe *)

				BitAppoggioPump_1:= NOT BitAppoggioPump_2					(* se la pompa 1 ha dei problemi *)
									AND NOT AllarmeHW_C1					(* Se non è presente l'allarme Salvamotore *)
									AND NOT AllarmeHW2_C1					(* Se non è presente l'allarme Contattore *)
									AND NOT PausaScambio.Q;					(* Finestra della pausa fra lo scambio delle pompe *)

			IF PumpA_AUTO THEN (* Con Pompa gestita in Automatico dal PLC *)
				IF CIR_STOP_REQ THEN
						 Pump_En[1] := FALSE;    (* solito gioco per forzare il Funzionemento della pompa da remoto il comando *)
				ELSIF CIR_RUN_REQ THEN
						Pump_En[1] := TRUE AND ScambioPompa;
				ELSE
					Pump_En[1]:=Delay.OUT AND BitAppoggioPump_1;
				END_IF
			END_IF

			IF PumpB_AUTO THEN
				IF CIR_STOP_REQ THEN
						 Pump_En[2] := FALSE;
				ELSIF CIR_RUN_REQ THEN
						Pump_En[2] := TRUE AND NOT ScambioPompa;
				ELSE
					Pump_En[2]:=Delay.OUT AND BitAppoggioPump_2;
				END_IF
			END_IF

ELSE
	mode:=1;

END_CASE


	Run:=Pump_En[1] OR Pump_En[2];

(* Set value on physical outuput! *)
PumpA_En := Pump_En[1];
PumpB_En := Pump_En[2];
END_ACTION

(* POU Plant_Objects/obj_CRON_EDITOR_01, ST *)
FUNCTION_BLOCK obj_CRON_EDITOR_01
(* === EDITOR CRONOGRAFO ===
   v1.0[16/04/15] - Versioning
   v1.1[19/05/15] - Create empty profile when not found
*)
VAR_INPUT

	(* Common selections *)
	CN_Sel:			BYTE:=1;
	CN_Act:			BYTE;
	CN_YSel:		WORD:=2015;
	CN_YAct:		WORD;

	(* Profile editor *)
	PR_Sel: 		BYTE:=1;
	PR_Act:			BYTE;
	PR_TT:			REAL;
	PR:				typ_Cron_Profile;
	(* Profile signals *)
	PR_Load:		BOOL;
	PR_Save:		BOOL;

	(* Calendar editor *)
	CA_Sel:			BYTE:=1; (* Calendar month selected *)
	CA_Act:			BYTE;    (* Calendar month active *)
	CA_DayF:		BYTE:=0;
	CA_DayL:		BYTE:=31;
	CA_TPR:			BYTE;
	CA:				typ_Cron_Calendar; (* Only used for first 32 entries *)
	(* Calendar signals *)
	CA_Load:		BOOL;
	CA_Save:		BOOL;

	(* Jolly editor *)
	JL:				ARRAY[0..9] OF typ_Cron_Jolly;
	(* Jolly signals *)
	JL_Load:		BOOL;
	JL_Save:		BOOL;

END_VAR
VAR_OUTPUT
	Message		: STRING;
END_VAR
VAR
	sFileName	: STRING;
	sFileMode	: STRING;
	hFile		: DWORD;
	Buf			: ARRAY[0..512] OF BYTE; (* AVOID THIS!! *)

	i			: WORD;
	ver			: BYTE;
	r1			: BOOL;
	r2			: DWORD;

	x: INT;
	maxProfili: INT;

	sFileNameOld	: STRING;
	sFileModeOld		: STRING;
	hFileOld			: DWORD;




	strAppoggio: STRING;
	FileGiaCreato: BOOL;
	fileCopiato: UDINT;

	tempMultiAnnoMax:INT;
	tempMultiAnnoIndex:INT;
	TEMP_MULTIANNO_MAX_DELTA:INT:=5;
	tempRicercaFileAnno:INT;
	tempAnno:INT;
	tempTrovato:BOOL;
END_VAR
IF PR_Load THEN PR_Load_Exe();
	PR_Load:=FALSE;
END_IF
IF PR_Save THEN
PR_Save_Exe();
PR_Save:=FALSE;
END_IF
IF CA_Load THEN
CA_Load_Exe();
CA_Load:=FALSE;
END_IF
IF CA_Save THEN
CA_Save_Exe();
CA_Save:=FALSE;
END_IF
IF JL_Load THEN
JL_Load_Exe();
JL_Load:=FALSE;
END_IF
IF JL_Save THEN
 JL_Save_Exe();
 JL_Save:=FALSE;
 END_IF
END_FUNCTION_BLOCK
ACTION CA_Load_Exe:
sFileMode:='r';
FileOpen();

IF hFile<>0 THEN

	(* Read calendar month *)
	FOR i := 0 TO 31 DO
		r1:=SysFileSetPos(File:=hFile, Pos:=(1024 + ((CA_Sel-1)*32 + i)*4));
		r2:=SysFileRead(File:=hFile, Buffer:=ADR(CA.Profile[i]), Size:=1);
	END_FOR

	(* Close file *)
	SysFileClose(File:=hFile);

	(* Validate data *)
	CA_Act :=CA_Sel;
	CN_Act :=CN_Sel;
	CN_YAct:=CN_YSel;

	Message:='Calendar load OK';

END_IF
END_ACTION
ACTION CA_Save_Exe:
sFileMode:='a';
FileOpen();

IF hFile<>0 THEN

	(* Write calendar month *)
	FOR i := 0 TO 31 DO
		r1:=SysFileSetPos(File:=hFile, Pos:=(1024 + ((CA_Sel-1)*32 + i)*4));
		r2:=SysFileGetPos(hFile);
		r2:=SysFileWrite(File:=hFile, Buffer:=ADR(CA.Profile[i]), Size:=1);
	END_FOR

	(* Close file *)
	SysFileClose(File:=hFile);

	Message:='Calendar save OK';

	(* db commentato! non salva i profili, ma solo il profilo corrente, che può anche essere modificato!*)
          (*PR_Save_exe();*)
	(* nel salvare il calendario aggiorno anche i profili così ho il file completo dei profili *)


END_IF

IF hFile<>0 THEN SysFileClose(File:=hFile); END_IF (*diego add*)
END_ACTION
ACTION FileOpen:
(* Create current filename 'yyyyCRnn.DAT' *) (* creo il nome del file da aparire *)
sFileName:=CONCAT(FilesPath,WORD_TO_STRING(CN_YSel));
sFileName:=CONCAT(STR1:=sFileName, STR2:='CR');
IF CN_Sel<10 THEN
sFileName:=CONCAT(STR1:=sFileName, STR2:='0');
END_IF
sFileName:=CONCAT(STR1:=sFileName, STR2:=BYTE_TO_STRING(CN_Sel));
sFileName:=CONCAT(STR1:=sFileName, STR2:='.DAT');


(* Apro il fiel in lettura per verificare se è presente altrimenti devo crearne uno nuovo a duplicare quello dell'anno precedente - apro 1  *)
hFile:=SysFileOpen(FileName:=sFileName, Mode:='r');
FileGiaCreato:=FALSE;

tempAnno:=CN_YSel;
tempTrovato:=FALSE;

(* File non trovato da creare  *)
IF hFile=0 THEN

	 (*cerco i file precendti: dall'anno prima fino a - TEMP_MULTIANNO_MAX_DELTA*)
	 tempRicercaFileAnno:=1;

	WHILE tempRicercaFileAnno<=TEMP_MULTIANNO_MAX_DELTA AND NOT tempTrovato DO


		strAppoggio:=INT_TO_STRING(tempAnno);
		(* Verifico se esite un file da cui partire *)
		StrAppoggio:=WORD_TO_STRING(STRING_TO_WORD(strAppoggio)-tempRicercaFileAnno);
		sFileNameOld:=CONCAT(FilesPath,StrAppoggio);

		sFileNameOld:=CONCAT(STR1:=sFileNameOld, STR2:='CR');
		IF CN_Sel<10 THEN
			sFileNameOld:=CONCAT(STR1:=sFileNameOld, STR2:='0');
		END_IF
		sFileNameOld:=CONCAT(STR1:=sFileNameOld, STR2:=BYTE_TO_STRING(CN_Sel));
		sFileNameOld:=CONCAT(STR1:=sFileNameOld, STR2:='.DAT');

		(* Apro il file in lettura per la verifica della presenza del file da copiare  *)
		hFileold:=SysFileOpen(FileName:=sFileNameOld, Mode:='r');

		IF hFileold<>0 THEN

			tempTrovato:=TRUE;

			fileCopiato:=SysFileCopy(sFileName,sFileNameold);

    		   	FileGiaCreato:=fileCopiato<>0;

			IF FileGiaCreato THEN
				Message:='File Sorgente/copia  trovato - file Copiato';
			ELSE
				Message:='File Sorgente/copia  trovato - file NON Copiato';
			END_IF


			(* Chiudo il file aperto per la verifica del file presente *)
			SysFileClose(File:=hFile);
			(* Chiudo il file aperto in lettura per la verifica della presenza del file da copiare  *)
			SysFileClose(File:=hFileold);

		END_IF

		tempRicercaFileAnno:=tempRicercaFileAnno+1;

	END_WHILE

	(* se non ho trovato nessun file..lo creo vuoto*)
	IF tempTrovato=FALSE THEN   (* file non trovato quindi devo crearne uno nuovo *)

			(* Create empty file *)
			hFile:=SysFileOpen(FileName:=sFileName, Mode:='w');
			MEMCLR(pDestinationAddress:=ADR(Buf), BytesToClear:=SIZEOF(Buf));
			FOR i := 0 TO 10239 BY 512 DO
				SysFileWrite(File:=hFile, Buffer:=ADR(Buf), Size:=512);
			END_FOR

			Buf[0]:=1;
			SysFileSetPos(File:=hFile, Pos:=0);
			SysFileWrite(File:=hFile, Buffer:=ADR(Buf), Size:=1);

			(* Chiudo il file aperto per la verifica del file presente *)
			SysFileClose(File:=hFile);
			(* Chiudo il file aperto in lettura per la verifica della presenza del file da copiare  *)
			SysFileClose(File:=hFileold);

			Message:='File Sorgente/copia non trovato-file Vuoto';

	END_IF


ELSE

	(* Chiudo il file aperto per la verifica del file presente *)
	SysFileClose(File:=hFile);

END_IF




(* Apro il file per permettere la scrittura o la lettura del file da parte delle altre action . la chiusura del file è delegata alle Action *)
hFile:=SysFileOpen(FileName:=sFileName, Mode:=sFileMode);
END_ACTION
ACTION JL_Load_Exe:
sFileMode:='r';
FileOpen();

IF hFile<>0 THEN

	(* Read jolly *)
	r1:=SysFileSetPos(File:=hFile, Pos:=512);
	r2:=SysFileRead(File:=hFile, Buffer:=ADR(JL), Size:=SIZEOF(JL));

	(* Close file *)
	SysFileClose(File:=hFile);

	(* Validate data *)
	CN_Act:=CN_Sel;
	CN_YAct:=CN_YSel;

	Message:='Jolly load OK';

END_IF
END_ACTION
ACTION JL_Save_Exe:
sFileMode:='a';
FileOpen();

IF hFile<>0 THEN

	(* Write selected profile *)
	r1:=SysFileSetPos(File:=hFile, Pos:=512);
	r2:=SysFileWrite(File:=hFile, Buffer:=ADR(JL), Size:=SIZEOF(JL));

	(* Close file *)
	SysFileClose(File:=hFile);

	Message:='Jolly save OK';

END_IF
END_ACTION
ACTION PR_Load_Exe:
sFileMode:='r';
FileOpen();

IF hFile<>0 THEN

	(* Read selected profile *)
	r1:=SysFileSetPos(File:=hFile, Pos:=(3072 + 512*PR_Sel));
	r2:=SysFileRead(File:=hFile, Buffer:=ADR(PR), Size:=SIZEOF(PR));

	(* Close file *)
	SysFileClose(File:=hFile);

	(* Validate data *)
	PR_Act:=PR_Sel;
	CN_Act:=CN_Sel;
	CN_YAct:=CN_YSel;

	Message:='Profile load OK';

END_IF
END_ACTION
ACTION PR_Save_Exe:
sFileMode:='a';
FileOpen();

IF hFile<>0 THEN

		(* Write selected profile *)
		r1:=SysFileSetPos(File:=hFile, Pos:=(3072 + 512*PR_Sel));
		r2:=SysFileWrite(File:=hFile, Buffer:=ADR(PR), Size:=SIZEOF(PR));

		(* Close file *)
		SysFileClose(File:=hFile);

		Message:='Profile save OK';

END_IF

IF hFile<>0 THEN SysFileClose(File:=hFile); END_IF (*diego add*)
END_ACTION
ACTION PR_Save_Exe_Multi:
(*eseguo  salvataggio profilo per l'anno corrente del CronoEditor - quello indicato da CN_YSel*)
CronEd.PR_Save_Exe();

(*verifico se esistono i file di schedulazioni per anni successivi: se aggiorno i profili anche lì*)

(*tempMultiAnnoMax dice fino a quale anno si considera*)
tempMultiAnnoMax:=CronEd.CN_YSel+TEMP_MULTIANNO_MAX_DELTA;

(* per ogni anno, vrifico se esiste il relativo file e se si aggiorno i profili anche li *)
FOR tempMultiAnnoIndex:=CronEd.CN_YSel+1 TO tempMultiAnnoMax BY 1 DO

	sFileName:=CONCAT(FilesPath,INT_TO_STRING(tempMultiAnnoIndex));
	sFileName:=CONCAT(STR1:=sFileName, STR2:='CR');
	IF CN_Sel<10 THEN
		sFileName:=CONCAT(STR1:=sFileName, STR2:='0');
	END_IF
	sFileName:=CONCAT(STR1:=sFileName, STR2:=INT_TO_STRING(CN_Sel));
	sFileName:=CONCAT(STR1:=sFileName, STR2:='.DAT');

	hFile:=SysFileOpen(FileName:=sFileName, Mode:='r');
	(* file esiste, aggiorno profili per quell'anno *)
	IF hFile<>0 THEN

		SysFileClose(File:=hFile);
		CronEd.CN_YSel:=tempMultiAnnoIndex;
		CronEd.PR_Save_Exe();

	ELSE
		SysFileClose(File:=hFile);

	END_IF


END_FOR
END_ACTION

(* POU Plant_Objects/obj_CRONTER_01, ST *)
FUNCTION_BLOCK obj_CRONTER_01
(* === THERMOSTAT ===
   v1.0[30/07/15] - Versioning
*)
VAR_INPUT
	(* Settings *)
	ID			: BYTE;		(* Index of instanced object *)

	InitOK		: BOOL;
	Alarm		: BOOL;
	Warning		: BOOL;

	Profile		: typ_Cron_Profile; 				(* Profilo attivo *)
	ProfileNr	: BYTE;								(* Indice profilo attivo *)
	CalendarIdx : WORD;								(* Indice calendario attivo *)
	Jolly		: ARRAY[0..9] OF typ_Cron_Jolly;	(* Jolly attivi *)

	Temperature	: INT;
	Local_MaxRunTAmb	:	INT;					(* Local maximum environment temperature, NOT "TAMB" *)
	Histeresys:INT; (* isteresi per la ripartenza del Comando ON*)


	sFile: 	STRING;


END_VAR
VAR_IN_OUT
END_VAR
VAR_OUTPUT
	SetPoint		: INT;
	Run				: BOOL;
	AntifreezeForce	: BOOL;
	RunCrono		: BOOL;

	(* Status *)
	Status_Log		: BYTE;
	Status_Vis 		: DWORD;
END_VAR
VAR
	Buf: 	ARRAY[0..512] OF BYTE; (* AVOID THIS!! *)
	hFile: 	DWORD;

	sFile2: STRING;

	i:		WORD;
	t1:		DWORD;
	t2:		BOOL;

END_VAR
(* Check initialization *)
(*IF NOT InitOK THEN Init(); END_IF*)

(* Check Temperature *)
IF Temperature <Local_MaxRunTAmb THEN

	(* LOCAL environment temperature lower than maximum allowed -> Proceed with SetPoint adjustment *)
	(* Chrono *)
(*	IF CalendarIdx<>Sys.Time_CT_Day THEN DB_Load(); END_IF *)

	IF CalendarIdx<>Sys.Time_CT_Day OR InitOK=FALSE THEN  (* col cambio della data carico il file corretti dove è intergrato il controllo della presenza del file *)
		CronEd(CN_Sel:=WORD_TO_BYTE(id),CN_YSel:=Sys.Time_Year, CA_Load:=TRUE,PR_Load:=TRUE);
		DB_Load(	sFile:= CronEd.sFileName);  (* aggiorno il SetPoint  partendo dal file noto*)
		InitOK:=TRUE;
	END_IF


	SetPoint:=Profile.Setpoint[Sys.Time_CT_Quarter];

	(* Check jolly *)
	FOR i := 0 TO 9 DO
		IF ( DT_TO_DWORD(Jolly[i].Start)>0  AND Jolly[i].End>Jolly[i].Start AND
		     Jolly[i].Start<=Sys.Time_CT_DT AND Jolly[i].End>Sys.Time_CT_DT ) THEN
				SetPoint:=Jolly[i].Temp;
		END_IF
	END_FOR

(*
	IF SetPoint < 180 THEN
		(* Switch off the device *)
		Run := FALSE;
	ELSE
		(* Set according to feedback T - Histeresys of 1°C *)
		IF Temperature >= (SetPoint + 5) THEN
			Run := FALSE;
		ELSIF Temperature <= (SetPoint - 5) THEN
			Run := TRUE;
		END_IF

		(* Between "SetPoint-5" and "SetPoint+5" last state (ON or OFF) of "Run" is kept	*)
	END_IF
*)
(* Gestione uscita Crono *)
		IF SetPoint>0 THEN RunCrono := TRUE;
		ELSIF SetPoint=0 THEN RunCrono := FALSE;
		END_IF

(* GEstione uscita Cronotermostato *)

		IF Temperature >= (SetPoint) THEN
			Run := FALSE;
		ELSIF Temperature <= (SetPoint - Histeresys) THEN
			Run := TRUE;
		END_IF
ELSE
	(* Environment overtemperature: stop heating -> Stop device *)
	Run := FALSE;
END_IF

(* Freeze warning: Switch on and heat! *)
(*IF Temperature < Plant_AntiFreezeTAmb THEN AntifreezeForce := TRUE;
ELSE AntifreezeForce := FALSE;
END_IF*)



(* Status color *)
   IF Alarm   THEN Status_Log:=2; Status_Vis:=COLOR_RED;
ELSIF Warning THEN Status_Log:=1; Status_Vis:=COLOR_YELLOW;
              ELSE Status_Log:=0; Status_Vis:=COLOR_GREEN;
			  END_IF
END_FUNCTION_BLOCK
ACTION AddLogData:
Logger.s1:=INSERT('&THER=',BYTE_TO_STRING(ID),5);
IF ID<10 THEN Logger.s1:=INSERT(Logger.s1,'0',5); END_IF

Logger.s1:=CONCAT(Logger.s1,INT_TO_STRING(SetPoint));			Logger.s1:=CONCAT(Logger.s1,';');

Logger.s1:=CONCAT(Logger.s1,WORD_TO_STRING(Status_Log));
ADDSTRING(ADR(Logger.TData), ADR(Logger.s1), Logger.TLen);
END_ACTION
ACTION DB_Create:
(* Create empty file *)
hFile:=SysFileOpen(FileName:=sFile, Mode:='w');

MEMCLR(pDestinationAddress:=ADR(Buf), BytesToClear:=SIZEOF(Buf));
FOR i := 0 TO 10239 BY 512 DO
	t1:=SysFileWrite(File:=hFile, Buffer:=ADR(Buf), Size:=512);		(* Clear created file (all bytes 0) *)
END_FOR
Buf[0]:=1;
t2:=SysFileSetPos(File:=hFile, Pos:=0);
t1:=SysFileWrite(File:=hFile, Buffer:=ADR(Buf), Size:=1);
SysFileClose(File:=hFile);
END_ACTION
ACTION DB_Load:
(*

DB_SetName();


(* File not found *)
IF hFile=0 THEN
	Warning:=TRUE;
	LogEv(EL_Wrn,EO_CRON,ID,1,'No_data_file');
	DB_Create();
	(* Reopen file *)
	hFile:=SysFileOpen(FileName:=sFile, Mode:='r');
	IF hfile=0 THEN
		Alarm:=TRUE;
		LogEv(EL_Alarm,EO_CRON,ID,3,'Filesystem_error');
		RETURN;
	END_IF
END_IF
*)

(* Open data file *)
hFile:=SysFileOpen(FileName:=sFile, Mode:='r');

(* Check version *)
SysFileRead(File:=hFile, Buffer:=ADR(Buf), Size:=1);
IF Buf[0]<>1 THEN
	IF NOT Alarm THEN
		Alarm:=TRUE;
		LogEv(EL_Alarm,EO_CRON,ID,2,'Bad_data_version');
	END_IF
	SysFileClose(File:=hFile);
	RETURN;
END_IF

(* Read Jolly data *)
t2:=SysFileSetPos(File:=hFile, Pos:=512);
t1:=SysFileRead(File:=hFile, Buffer:=ADR(Jolly), Size:=SIZEOF(Jolly));
(* Read active profile index *)
CalendarIdx:=Sys.Time_CT_Day;
t2:=SysFileSetPos(File:=hFile, Pos:=(1024+4*CalendarIdx));
t1:=SysFileRead(File:=hFile, Buffer:=ADR(ProfileNr), Size:=SIZEOF(ProfileNr));
(* Read active profile *)
t2:=SysFileSetPos(File:=hFile, Pos:=(3072+512*ProfileNr));
t1:=SysFileRead(File:=hFile, Buffer:=ADR(Profile), Size:=SIZEOF(Profile));

(* Close file and validate data *)
SysFileClose(File:=hFile);
END_ACTION
ACTION DB_SetName:
(* Create current filename 'yyyyCRnn.DAT' *)
sFile:=CONCAT(FilesPath,WORD_TO_STRING(Sys.Time_Year));
sFile:=CONCAT(STR1:=sFile, STR2:='CR');
IF ID<10 THEN
sFile:=CONCAT(STR1:=sFile, STR2:='0');
END_IF
sFile:=CONCAT(STR1:=sFile, STR2:=BYTE_TO_STRING(ID));
sFile:=CONCAT(STR1:=sFile, STR2:='.DAT');
END_ACTION
ACTION Init:
DB_Load();
InitOK:=TRUE;
END_ACTION

(* POU Plant_Objects/obj_EV_01, ST *)
FUNCTION_BLOCK obj_EV_01
(* === CIRCOLATORE GEMELLARE STANDARD ===
   VERSIONE 01 REALIZZATA DA MORENO E TESTA SU IMPIANTO SAN FELICE ID 003 CLV
*)

VAR_INPUT
	(* Settings *)
	ID				: BYTE;
	(* Physical inputs (Force) *)
	EV_OPEN_REQ		: BOOL; (* External run request (no heat or cold requested) *)
	EV_CLOSE_REQ	: BOOL; (* External stop request (has priority over RUN signals!) *)

	(* Physical inputs (Feedback) *)
	EV_Open			: BOOL; (* Micro switch esegnalazione elttrovalvola Aperta *)
	EV_Close		: BOOL; (* Micro Switch segnalazione elettrovalvola Chiusa *)
	EV_Auto			: BOOL; (* Micro Switch segnalazione elettrovalvola Chiusa *)



	Mod_ComandoEV	: BOOL :=FALSE ; (* bit che stabilisce che tipo di comanda dare:
										con Mod_ComandoEV=0 la valvola è NC con comando a 1 si apre, 
										con Mod_ComandoEV=1	la valvola è NO con comando a 1 si chiude  *)

	(* Controlllo *)
	OnOff			: BOOL;	(* On/Off da cronotermostato a da abilitazione esternao *)

	(* Working mode: 0-Both pumps works simultaneously, 1-Alternate every 24h, 2-Master/Backup *)
	InitOK			: BOOL;


END_VAR
VAR_OUTPUT
	EV_En			: BOOL; (* Comando in uscita *)

	Ctrl_Run		:	BOOL;		(* Logical status of the device: 0: Not running (switched off), 1: running *)
	Run				:	BOOL;		(* Real status *)

	Status_Log		: WORD;
	Status_Vis		: DWORD;
END_VAR
VAR

	(* Filters *)
	fEV_ST_OPEN		: 	FLT_TIME := (INITEV:=FALSE,TTAP:=T#35s);
	fEV_ST_CLOSE	: 	FLT_TIME := (INITEV:=FALSE,TTAP:=T#35s);
	fEV_AUTO		:	FLT_TAP;

	(* Timer manage switch on/off delay *)
	Delay		: 	TONOF;

	(* Alarm and Warning counters *)
	AllarmeHW_EV_Open: BOOL;
	AllarmeHW_EV_Close: BOOL;

	WarningEV_inMan:BOOL;

	CHECK_OPEN: BOOL;
	CHECK_CLOSE: BOOL;
END_VAR
VAR_INPUT RETAIN

	(* Timings *)
	OnDelay		:	TIME;	(* Switch on delay *)
	OffDelay	:	TIME;	(* Switch off delay *)

END_VAR
Init();

EV_Manager();

(* Check alarms and warnings *)
CheckFault();

IF ( AllarmeHW_EV_Open ) OR  ( AllarmeHW_EV_Close) THEN
	Status_Log := 2;
	Status_Vis := COLOR_RED;
ELSIF
	WarningEV_inMan THEN
	Status_Log := 1;
	Status_Vis := COLOR_YELLOW;
ELSE
	Status_Log := 0;
	Status_Vis := COLOR_GREEN;
END_IF
END_FUNCTION_BLOCK
ACTION AddLogData:
Logger.s1:=INSERT('&EV=',BYTE_TO_STRING(ID),3);
IF ID<10 THEN Logger.s1:=INSERT(Logger.s1,'0',3); END_IF

Logger.s1:=CONCAT(Logger.s1,SEL(EV_En,'0','1'));
Logger.s1:=CONCAT(Logger.s1,';');
Logger.s1:=CONCAT(Logger.s1,SEL(EV_Open,'0','1'));
Logger.s1:=CONCAT(Logger.s1,';');
Logger.s1:=CONCAT(Logger.s1,SEL(EV_Close,'0','1'));
Logger.s1:=CONCAT(Logger.s1,';');
Logger.s1:=CONCAT(Logger.s1,WORD_TO_STRING(Status_Log));
Logger.s1:=CONCAT(Logger.s1,';');
Logger.s1:=CONCAT(Logger.s1,SEL(EV_OPEN_REQ,'0','100'));
Logger.s1:=CONCAT(Logger.s1,';');
Logger.s1:=CONCAT(Logger.s1,SEL(EV_CLOSE_REQ,'0','100'));


ADDSTRING(ADR(Logger.TData), ADR(Logger.s1), Logger.TLen);
END_ACTION
ACTION CheckFault:
(*** ALARMS ***)

(**** Elettrovalvola non si Apre ****)
(* Allarme Hardware da ingresso PLC *)

 (* bit che stabilisce che tipo di comanda dare: con Mod_ComandoEV=0 la valvola è NC con comando a 1 si apre,
												con Mod_ComandoEV=1	la valvola è NO con comando a 1 si chiude  *)
IF Mod_ComandoEV THEN

	CHECK_OPEN:=(EV_EN AND NOT EV_Open);
	fEV_ST_OPEN(IN:=CHECK_OPEN);
	IF fEV_ST_OPEN.EVH THEN
		LogEv(EL_Alarm,EO_EV,ID,3,'MancataApertura');
		AllarmeHW_EV_Open := TRUE;
	END_IF

	IF AllarmeHW_EV_Open AND EV_Open THEN
		LogEv(EL_Log,EO_EV,ID,4,'ElettrovalvolaRiaperta');
		AllarmeHW_EV_Open := FALSE;
	END_IF

	(**** Elettrovalvola non si chiude ****)
	(* Allarme Hardware da ingresso PLC *)

	CHECK_CLOSE:=(NOT EV_EN AND NOT EV_Open);

	fEV_ST_CLOSE(IN:=CHECK_CLOSE);
	IF fEV_ST_CLOSE.EVH THEN
		LogEv(EL_Alarm,EO_EV,ID,5,'MancataChiusura');
		AllarmeHW_EV_CLose := TRUE;
	END_IF

	IF AllarmeHW_EV_CLose AND EV_close THEN
		LogEv(EL_Log,EO_EV,ID,6,'ElettrovalvolaRichiusa');
		AllarmeHW_EV_CLose := FALSE;
	END_IF
ELSE
	CHECK_OPEN:=NOT EV_EN AND NOT EV_Open;
	fEV_ST_OPEN(IN:=CHECK_OPEN);
	IF fEV_ST_OPEN.EVH THEN
		LogEv(EL_Alarm,EO_EV,ID,3,'MancataApertura');
		AllarmeHW_EV_Open := TRUE;
	END_IF

	IF AllarmeHW_EV_Open AND EV_Open THEN
		LogEv(EL_Log,EO_EV,ID,4,'ElettrovalvolaRiaperta');
		AllarmeHW_EV_Open := FALSE;
	END_IF

	(**** Elettrovalvola non si chiude ****)
	(* Allarme Hardware da ingresso PLC *)

	CHECK_CLOSE:=EV_EN AND NOT EV_close;

	fEV_ST_CLOSE(IN:=CHECK_CLOSE);
	IF fEV_ST_CLOSE.EVH THEN
		LogEv(EL_Alarm,EO_EV,ID,5,'MancataChiusura');
		AllarmeHW_EV_CLose := TRUE;
	END_IF

	IF AllarmeHW_EV_CLose AND EV_close THEN
		LogEv(EL_Log,EO_EV,ID,6,'ElettrovalvolaRichiusa');
		AllarmeHW_EV_CLose := FALSE;
	END_IF

END_IF

(* Verify if in Auto or Manual mode *)
fEV_AUTO(IN:=EV_AUTO);
(*** Pump A ***)
IF fEV_AUTO.EVH THEN
	LogEv(EL_Log,EO_EV,ID,1,'Elettrovalvola_in_AUTOMATIC_MODE');
	WarningEV_inMan := FALSE;
END_IF

(* Manual -> Keep switched on *)
IF fEV_AUTO.EVL THEN
	LogEv(EL_Wrn,EO_EV,ID,2,'Elettrovalvola_in_MANUAL_MODE');
	WarningEV_inMan := TRUE;
END_IF
END_ACTION
ACTION EV_Manager:
(* Verify if OnOff is changed *)
Ctrl_Run := OnOff;

(* Check switch on or switch off delay *)

IF OffDelay<t#1s THEN
	 OffDelay:=t#10m0s;
END_IF;

Delay(IN:=Ctrl_Run,PT_OF:=OffDelay,PT_ON:=OnDelay + WORD_TO_TIME(1000*ID));    (* Ritardo all'accensione e allo Spegnimento *)


IF Mod_ComandoEV THEN
	IF EV_AUTO THEN
		IF EV_CLOSE_REQ THEN
			EV_En := FALSE;
		ELSIF
			EV_OPEN_REQ THEN EV_En := TRUE;
		ELSE
			EV_En:= Delay.OUT;
		END_IF
	END_IF
ELSE
	IF EV_AUTO THEN
		IF EV_CLOSE_REQ THEN
			EV_En := TRUE;
		ELSIF
			EV_OPEN_REQ THEN EV_En := FALSE;
		ELSE
			EV_En:= NOT Delay.OUT;
		END_IF
	END_IF
END_IF



Run:=EV_En;
END_ACTION
ACTION Init:
IF NOT InitOK THEN

	EV_EN := FALSE;
	InitOK := TRUE;

END_IF
END_ACTION

(* POU Plant_Objects/obj_GAS, ST *)
FUNCTION_BLOCK obj_GAS
(* === GENERIC PULSE GAS CONTABILIZER ===
   v1.0[23/03/15] - Cleanup and logger action
*)
VAR_INPUT
	(* Settings *)
	ID				: BYTE;			(* Index of instanced object *)
	Peso			: INT:=1;		(* Weight of inpulse [m^3] *)
	TempoTimeOut	: TIME:=T#1m;	(* Activity timeout for warning *)
	(* Physical inputs *)
	GAS_DI			: BOOL;	(* Pulse digital input *)
END_VAR
VAR_IN_OUT
	Contatore       : DINT;
	Totalizzatore	: DINT; (* Totale Conteggio x valore peso *)
END_VAR
VAR_OUTPUT
	(* Status *)
	Status_Log		: BYTE;
	Status_Vis 		: DWORD;
END_VAR
VAR
	Counter			: FLT_TAP := (TAP:=2);
	TimeOut			: TON;
	Warning			: FLT_EVENT;
END_VAR
(* Imposto il time out se non c'è movimento sulla linea per il tempo impostato loggo un Warning *)
TimeOut( IN:=NOT GAS_DI, PT:=TempoTimeOut );

Warning( IN:= TimeOut.Q );

IF Warning.EVH THEN
	(* Condizione di WARNING *)
	Status_Log:=1; Status_Vis:=COLOR_YELLOW;
	LogEv(EL_Wrn,EO_GAS,ID,2,'Nessun_Movimento');
END_IF

IF Warning.EVL THEN
	(* Condizione di Rientro dal WARNING *)
	Status_Log:=0; Status_Vis:=COLOR_GREEN;
	LogEv(EL_Log,EO_GAS,ID,1,'');
END_IF
END_FUNCTION_BLOCK
ACTION Count:
(* Triggero sul fronte di salita l'ingresso digitale *)
Counter(IN:=GAS_DI);

(* Conto i fronti di salita  in modo de creare rapporto*)
IF Counter.EVH THEN
	Contatore:=Contatore+1;
	Totalizzatore:=Contatore*Peso;
END_IF
END_ACTION

(* POU Plant_Objects/obj_MBUS, ST *)
FUNCTION_BLOCK obj_MBUS
(* === M-BUS PROTOCOL INTERFACE ===
   v1.0[16/03/15] - Added interface errors
*)
VAR_INPUT
	(* Settings *)
	ID				: BYTE;
	COM				: BYTE;
	BAUDRATE		: COM_BAUDRATE;
	(* Interface *)
	MBus 			: typMBus;
	MBus_Master 	: FbMBusMaster;
END_VAR
VAR_OUTPUT
	(* Status *)
	Status_Log		: BYTE;
	Status_Vis 		: DWORD;
END_VAR
VAR
	Alarm			: FLT_EVENT;
END_VAR
MBus_Master( bCOMPORT:=COM , enumBAUDRATE:=BAUDRATE , utMBus:=MBus );

(* Check status *)
Alarm(IN:=(MBus.bCOM_ERROR<>0));
IF Alarm.EVH THEN
	LogEv(EL_Alarm,EO_MBUS,ID,1,BYTE_TO_STRING(MBus.bCOM_ERROR));
END_IF
IF Alarm.EVL THEN
	LogEv(EL_Log,EO_MBUS,ID,2,'MBUS_OK');
END_IF

(* Log/visu status *)
   IF Alarm.IN   					THEN Status_Log:=2; Status_Vis:=COLOR_RED;
ELSIF (MBus.bL1_ERROR AND 16#1F)<>0 THEN Status_Log:=1; Status_Vis:=COLOR_YELLOW;
  				 					ELSE Status_Log:=0; Status_Vis:=COLOR_GREEN;
END_IF
END_FUNCTION_BLOCK

(* POU Plant_Objects/obj_MBUS_CTB_SCANNER, ST *)
FUNCTION_BLOCK obj_MBUS_CTB_SCANNER
(* === MBUS HEAT CONTABILIZERS SCANNER & MANAGER ===
   v1.0[16/04/05] - Versioning
   v1.1[29/06/05] - Support for secondary addresses

	> Save/Load of CTB configuration on SD card 'CTBS01.DAT'

*)
VAR_INPUT
	(* Settings *)
	ID				: BYTE;
	EndScanAddress	: BYTE:=250;
	EndlessRescan   : BOOL:=FALSE;
	RefreshPause	: TIME:=t#240s; (* Refresh pause after complete reading cycle *)
	RescanPause		: TIME:=t#30s;  (* Scan pause after successful reading / refresh retry delay *)
	(* Controls *)
	Refresh			: BOOL; (* Enable automatic refresh of detected CTBs *)
	ListLoad		: BOOL:=TRUE; (* Load list from file *)
	ListSave		: BOOL; (* Save list to file *)
	Rescan			: BOOL; (* Perform complete search for list-update *)
END_VAR
VAR_IN_OUT
	MBUS			: obj_MBUS;
END_VAR
VAR_OUTPUT
(*	ConnectedCTBs	: BYTE; (* Number of connected CTBs at last rescan *)*)
	(* Status *)
	Status_Log		: BYTE;
	Status_Vis 		: DWORD;
END_VAR
VAR

	(* Virtual contabilizer for scanner *)
	M1			: FbMBus_Heat := (xSND_NKE:=FALSE);
	M1_Start	: BOOL;
	C1			: FbUnitConverter;
	C1_Err		: BOOL;

	(* Contabilizers data *)
	CTBS		: ARRAY [0..255] OF typ_MBUS_CTBS;

	sta			: BYTE; (* Status: 0:Idle, 1:Wait scan response, 2:Wait refresh response, 3:Wait refresh delay *)
	cnt		 	: BYTE; (* Selection counter *)
	retry		: BYTE; (* Retries counter *)
	pass_cnt 	: BYTE; (* Active counter *)
	dly 	 	: TON;
	s1 		 	: STRING;

	hName	 : STRING;
	hFile	 : DWORD;
	hOK		 : BOOL;
	hCnt	 : BYTE;

END_VAR
CASE sta OF
	0: (*** INIT ***)
		hName:=INSERT('CTBS.DAT',BYTE_TO_STRING(ID),4);
		IF ID<10 THEN hName:=INSERT(hName,'0',4); END_IF
		hName:=CONCAT(FilesPath,hName);
		sta:=1;

	1: (*** Wait actions ***)
		(* Check load request *)
		IF ListLoad THEN
			ListLoad:=FALSE;
			ListLoad_Exe();
			IF hOK THEN
				Refresh:=TRUE;
			END_IF
		END_IF
		(* Check save request *)
		IF ListSave THEN
			ListSave:=FALSE;
			ListSave_Exe();
		END_IF
		(* Check MBUS not busy *)
		IF NOT M1_Start THEN
			IF Rescan THEN
				(* Start scanning - with fast timeout and only one retry *)
				cnt:=0;
				pass_cnt:=0;
				MBUS.MBus_Master.bRetries:=1;
				MBUS.MBus_Master.tTimeout:=T#1000ms;
				M1.dwAdr:=cnt;
				M1_Start:=TRUE;
				CTBS[cnt].Status_Vis:=COLOR_LBLUE;
				sta:=10;
			ELSIF Refresh THEN
				(* Start refresh *)
				cnt:=0;
				retry:=0;
				GoToNextActive();
				IF cnt>EndScanAddress THEN
					Refresh:=FALSE;
				ELSE
					MBUS.MBus_Master.bRetries:=1;
					MBUS.MBus_Master.tTimeout:=T#2000ms;
					M1.dwAdr:=CTBS[cnt].Address;
					M1_Start:=TRUE;
					sta:=20;
				END_IF
			END_IF
		END_IF

	10: (*** PRIMARY SCAN ***)
		IF NOT Rescan THEN
			sta:=1;
		ELSE
			IF NOT M1_Start THEN
				(* Get scan result *)
				UpdateNode();
				(* Next object *)
				cnt:=cnt+1;
				IF cnt>EndScanAddress THEN
					(*ConnectedCTBs:=pass_cnt;*)
					Rescan:=EndlessRescan;
					sta:=1;
				ELSE
					IF CTBS[cnt-1].Present THEN
						(*dly(IN:=FALSE, PT:=RescanPause);*)
						sta:=11;
					ELSE
						M1.dwAdr:=cnt;
						M1_Start:=TRUE;
						CTBS[cnt].Status_Vis:=COLOR_LBLUE;
					END_IF
				END_IF
			END_IF
		END_IF

	11: (*** PRIMARY SCAN DELAY ***)
		dly(IN:=NOT dly.Q, PT:=RescanPause);
		IF dly.Q THEN
			M1.dwAdr:=cnt;
			M1_Start:=TRUE;
			sta:=10;
		END_IF

	20: (*** REFRESH CTBs READING *)
		IF (NOT Refresh) OR Rescan THEN
			sta:=1;
		ELSE
			IF NOT M1_Start THEN
				(* Check result *)
				IF M1.bError<>0 AND retry<2 THEN
					retry:=retry+1;
					sta:=22;
				ELSE
					(* Get scan result *)
					UpdateNode();
					(* Next object *)
					cnt:=cnt+1;
					GoToNextActive();
					retry:=0;
					IF cnt>EndScanAddress THEN
						sta:=21;
						(*dly(IN:=FALSE, PT:=RefreshPause);*)
					ELSE
						M1.dwAdr:=CTBS[cnt].Address;
						M1_Start:=TRUE;
					END_IF
				END_IF
			END_IF
		END_IF

	21: (*** REFRESH CTBs READING - CYCLE PAUSE ***)
		dly(IN:=NOT dly.Q, PT:=RefreshPause);
		IF dly.Q THEN sta:=1; END_IF

	22: (*** REFRESH CTBs READING - RETRY PAUSE ***)
		dly(IN:=NOT dly.Q, PT:=RescanPause);
		IF dly.Q THEN M1_Start:=TRUE; sta:=20; END_IF

ELSE
	sta:=0;
END_CASE

(* Update virtual contabilizer *)
M1( utMBus:=MBUS.MBus , xStart:=M1_Start );
END_FUNCTION_BLOCK
ACTION AddLogData:
;(*
FOR Logger.i1 := 0 TO EndScanAddress  DO
	IF 	CTBSCAN01.NodoMBusPresente[Logger.i1]=TRUE THEN
		Logger.s1:=INSERT('&CTB=',WORD_TO_STRING(Logger.i1),4);
		IF Logger.i1<10 THEN Logger.s1:=INSERT(Logger.s1,'0',4); END_IF
	    Logger.s1:=CONCAT(Logger.s1,'0' (*CTBSCAN01.CTB_utFTemp [Logger.i1].Value*) ); Logger.s1:=CONCAT(Logger.s1,';');
		Logger.s1:=CONCAT(Logger.s1,'0' (*CTBSCAN01.CTB_utRTemp [Logger.i1].Value*) ); Logger.s1:=CONCAT(Logger.s1,';');
		Logger.s1:=CONCAT(Logger.s1,'0' (*CTBSCAN01.CTB_utFlow  [Logger.i1].Value*) ); Logger.s1:=CONCAT(Logger.s1,';');
		Logger.s1:=CONCAT(Logger.s1,'0' (*CTBSCAN01.CTB_utPower [Logger.i1].Value*) ); Logger.s1:=CONCAT(Logger.s1,';');
		Logger.s1:=CONCAT(Logger.s1,'0' (*CTBSCAN01.CTB_utEnergy[Logger.i1].Value*) ); Logger.s1:=CONCAT(Logger.s1,';');
		Logger.s1:=CONCAT(Logger.s1,BYTE_TO_STRING(CTBSCAN01.Status_Log_NodoMBus[Logger.i1]));
		ADDSTRING(ADR(Logger.TData), ADR(Logger.s1), Logger.TLen);
	END_IF
END_FOR
*)
END_ACTION
ACTION GoToNextActive:
WHILE CTBS[cnt].Present <> TRUE AND cnt<=EndScanAddress DO
	cnt:=cnt+1;
END_WHILE
END_ACTION
ACTION ListLoad_Exe:
hOK:=FALSE;
hFile:=SysFileOpen(hName,'r');
IF hFile<>0 THEN
	FOR hCnt := 1 TO EndScanAddress  DO
		SysFileRead(hFile, ADR(CTBS[hCnt].Present), SIZEOF(CTBS[hCnt].Present));
		SysFileRead(hFile, ADR(CTBS[hCnt].Address), SIZEOF(CTBS[hCnt].Address));
		CTBS[hCnt].Status_Vis:=SEL(CTBS[hCnt].Present,COLOR_GREY,COLOR_LBLUE);
	END_FOR
	SysFileClose(hFile);
	hOK:=TRUE;
END_IF
END_ACTION
ACTION ListSave_Exe:
hOK:=FALSE;
hFile:=SysFileOpen(hName,'w');
IF hFile<>0 THEN
	FOR hCnt := 1 TO EndScanAddress  DO
		SysFileWrite(hFile, ADR(CTBS[hCnt].Present), SIZEOF(CTBS[hCnt].Present));
		SysFileWrite(hFile, ADR(CTBS[hCnt].Address), SIZEOF(CTBS[hCnt].Address));
	END_FOR
	SysFileClose(hFile);
	hOK:=TRUE;
END_IF
END_ACTION
ACTION UpdateNode:
(* Save node data *)
CTBS[cnt].NodeError:=M1.bError;
CTBS[cnt].Info:=M1.utMBInfo;
C1(utMBRecord:=M1.utFTemp  , utUnit:=C    , rValue=>CTBS[cnt].Data_FTemp  , xError=>C1_Err );
C1(utMBRecord:=M1.utRTemp  , utUnit:=C    , rValue=>CTBS[cnt].Data_RTemp  , xError=>C1_Err );
C1(utMBRecord:=M1.utFlow   , utUnit:=m3ph , rValue=>CTBS[cnt].Data_Flow   , xError=>C1_Err );
C1(utMBRecord:=M1.utPower  , utUnit:=W    , rValue=>CTBS[cnt].Data_Power  , xError=>C1_Err );
C1(utMBRecord:=M1.utEnergy , utUnit:=kWh  , rValue=>CTBS[cnt].Data_Energy , xError=>C1_Err );

(* Check node status *)
IF CTBS[cnt].NodeError<>0  THEN
	(* se non sono in allarme di comunicazione loggo l'allarme *)
	IF CTBS[cnt].Status_Log<>2 AND sta=20 THEN
		LogEv(EL_Alarm,EO_CTB,cnt,2,CONCAT('Err',BYTE_TO_STRING(CTBS[cnt].NodeError)));
	END_IF
	(*Check rescan mode *)
	IF sta=10 THEN
		(* Disable presence flag & set grey status *)
		CTBS[cnt].Present:=FALSE;
		CTBS[cnt].Address:=0;
		CTBS[cnt].Status_Log:=3;
		CTBS[cnt].Status_Vis:=COLOR_GREY;
	ELSE
		(* Update status *)
		CTBS[cnt].Status_Log:=2;
		CTBS[cnt].Status_Vis:=COLOR_RED;
	END_IF
ELSE
	(* tutto OK Comunizaione andata a buon termine *)
	(* se non sono in allarme di comunicazione loggo l'allarme, ma  se non presente *)
	IF CTBS[cnt].Status_Log<>0 AND sta=20 THEN
		LogEv(EL_Log,EO_CTB,cnt,1,'Nodo_OK');
	END_IF
	(*se sono in fase di rescan memorizzo la presenza del nodo *)
	IF sta=10 THEN
		CTBS[cnt].Present:=TRUE;
		CTBS[cnt].Address:=cnt;
		pass_cnt:=pass_cnt+1;
	END_IF
	(* Update status *)
	CTBS[cnt].Status_Log:=0;
	CTBS[cnt].Status_Vis:=COLOR_GREEN;
END_IF

(* Send data to logger on refresh *)
IF sta=20 THEN
	Logger_Head();
		Logger.s1:=INSERT('&CTB=',WORD_TO_STRING(cnt),4);
		IF cnt<10 THEN Logger.s1:=INSERT(Logger.s1,'0',4); END_IF
	    Logger.s1:=CONCAT(Logger.s1, DINT_TO_STRING(REAL_TO_DINT(CTBS[cnt].Data_FTemp*10  )) ); Logger.s1:=CONCAT(Logger.s1,';');
		Logger.s1:=CONCAT(Logger.s1, DINT_TO_STRING(REAL_TO_DINT(CTBS[cnt].Data_RTemp*10  )) ); Logger.s1:=CONCAT(Logger.s1,';');
		Logger.s1:=CONCAT(Logger.s1, DINT_TO_STRING(REAL_TO_DINT(CTBS[cnt].Data_Flow*1000 )) ); Logger.s1:=CONCAT(Logger.s1,';');
		Logger.s1:=CONCAT(Logger.s1, DINT_TO_STRING(REAL_TO_DINT(CTBS[cnt].Data_Power     )) ); Logger.s1:=CONCAT(Logger.s1,';');
		Logger.s1:=CONCAT(Logger.s1, DINT_TO_STRING(REAL_TO_DINT(CTBS[cnt].Data_Energy/10 )) ); Logger.s1:=CONCAT(Logger.s1,';');
		Logger.s1:=CONCAT(Logger.s1, BYTE_TO_STRING(CTBS[cnt].Status_Log) );
		ADDSTRING(ADR(Logger.TData), ADR(Logger.s1), Logger.TLen);
	Logger_Send();
END_IF

(*VisuDatiMbus[cnt].sdNodoPresente :=SEL(NodoMBusPresente[cnt],'FAIL!','OK'); *)

(* Log found event during scan *)
IF sta=10 AND CTBS[cnt].Present THEN
	s1:='FOUND_';
	s1:=CONCAT(s1, CTBS[cnt].Info.stMED);
	s1:=CONCAT(s1,'_');
	s1:=CONCAT(s1, CTBS[cnt].Info.stID);
	LogEv(EL_Log,EO_CTB,cnt,100,s1);
END_IF
END_ACTION

(* POU Plant_Objects/obj_PORT, ST *)
FUNCTION_BLOCK obj_PORT
(* === FLOW&VOLUME CONTABILIZER ===
   v1.0[16/04/05] - Versioning
*)
VAR_INPUT
	(* Settings *)
	ID			: BYTE;
	Peso		 : INT:=1;		(* Peso dell' impulso , serve per avere una lettura immediata dell'unità ingegneristica *)
	TempoTimeOut : TIME;		(* Minuti di inattività per la segnalazione del WRN *)
	PuntoMinX	: DINT;			(*Parametri per la scalatura *)
	PuntoMaxX	: DINT;
	PuntoMinY	: REAL;
	PuntoMaxY	: REAL;

	TAP			: INT:=2000;   (* Filtro in msec *)
	INITEV		: BOOL:= TRUE; (* Generate init OK event *)
	SogliaHH	: WORD;    (* Soglia per segnalazione Allarme Extra Range in alto - Solitamente sondo in CC *)
	SogliaHL	: WORD;    (* Soglia per segnalazione Allarme Extra Range in Basso - Solitamente sondo Aperta *)
	SogliaWH	: REAL;    (* Soglia per segnalazione Warning  in alto  *)
	SogliaWL	: REAL;    (* Soglia per segnalazione Warning in basso  *)

	(* Physical inputs *)
	DI_INPUT	: BOOL;		(* Ingresso Digitale per il conteggio  *)
	AI_INPUT	: WORD;		(* Ingresso Analogico *)
END_VAR
VAR_IN_OUT
    Contatore		: DINT;
    Totalizzatore	: DINT; (* Totale Conteggio x valore peso *)
END_VAR
VAR_OUTPUT
	ValoreScalato	: DINT;	(* Valore istantaneo scalato ingresso Analgico *)
	ERR				: BOOL;	(* Segnalazione Errore *)
	WRN				: BOOL;	(* Segnalazione Warning *)
	(* Status *)
	Status_Log	: BYTE;
	Status_Vis 	: DWORD;
END_VAR
VAR
	TRig_DI			: R_TRIG;
	TimeOut			: TON;
	TRigR_TimeOut	: R_TRIG;
	TRigL_TimeOut	: F_TRIG;
	SegnaleHH		: BOOL;
	SegnaleHL		: BOOL;
	SegnaleOK		: BOOL;
	SegnaleWH		: BOOL;
	SegnaleWL		: BOOL;
	FiltroWRN		: TON;
	FiltroOK		: TON;
	FiltroERR		: TON;
END_VAR
(*****************************************************************************************)
(**** Gestione ingresso digitale per la contabilizzazzione degli impulsi *****************)
(*****************************************************************************************)

TRig_DI(CLK:=DI_Input );
IF  TRig_DI.Q THEN
	Contatore:=Contatore+1;
	Totalizzatore:=Contatore*Peso;
END_IF

(* Activity monitoring *)
TimeOut(IN:=NOT DI_Input , PT:=TempoTimeOut, Q=> , ET=> );
TRigR_TimeOut(CLK:= TimeOut.Q  );
TRigL_TimeOut(CLK:= TimeOut.Q  );

IF  TRigR_TimeOut.Q THEN
	WRN:=TRUE;
	LogEv(EL_Wrn,EO_PORT,ID,5,'Nessun_Movimento');
END_IF

IF  TRigL_TimeOut.Q THEN
	WRN:=FALSE;
	LogEv(EL_Log,EO_PORT,ID,1,'');
END_IF


(*****************************************************************************************)
(**** Gestione ingresso Analogico per la gestione del valore istantaneo  *****************)
(*****************************************************************************************)

(* Verifico che le variabile letta dall'ingresso Analogico  sia dentro i range
ATTENZIONE I LIMITI SPESSO SONO IN WORD VERIFICA  TABELLA MANUALE WAGO  *)
SegnaleHH:=(AI_INPUT>=SogliaHH);
SegnaleHL:=(AI_INPUT<=SogliaHL);
SegnaleOK:=NOT (SegnaleHH OR SegnaleHL);

(* Linerarizzo il segnale di ingresso e la converto in unita ingegneristiche *)
ValoreScalato:=REAL_TO_DINT(LINEAR( AI_INPUT, PuntoMinY, PuntoMinX, PuntoMaxY, PuntoMaxX ));


IF SegnaleOK  THEN
	(*  Verifica  e segnalazione Warning *)
	SegnaleWH:=(ValoreScalato>SogliaWH);
	SegnaleWL:=(ValoreScalato<SogliaWL);

		FiltroWRN(IN:=(SegnaleWH OR SegnaleWL)  , PT:=INT_TO_TIME(TAP) );    (* Filtro su LOG *)
		IF  FiltroWRN.Q THEN     (* Condizione di WARNING *)
			IF NOT WRN THEN
				WRN:=TRUE;
 				LogEv(EL_Wrn,EO_PORT,ID,SEL(ValoreScalato<=SogliaWL,3,2),DINT_TO_STRING(ValoreScalato));
			END_IF
		END_IF

	IF (INITEV OR WRN OR ERR)  AND NOT FiltroWRN.Q THEN
		FiltroWRN(IN:=FALSE  , PT:=INT_TO_TIME(TAP));    (* Resetto il Filtro su LOG WRN  *)
		FiltroERR(IN:=FALSE  , PT:=INT_TO_TIME(TAP));    (* Resetto il Filtro su LOG ERR *)
		INITEV:=FALSE; ERR:=FALSE; WRN:=FALSE;
		LogEv(EL_Log,EO_PORT,ID,1,'');
	END_IF

	Status_Log:=0;
	Status_Vis:=16#20F020;
ELSE
		FiltroERR(IN:=TRUE , PT:= INT_TO_TIME(TAP) );    (* Filtro su LOG *)
			IF  FiltroERR.Q THEN     (* Condizione di WARNING *)
					IF NOT ERR THEN
						ERR:=TRUE;
						IF SegnaleHH THEN LogEv(EL_Alarm,EO_PORT,ID,6,DINT_TO_STRING(ValoreScalato));END_IF;
						IF SegnaleHL THEN LogEv(EL_Alarm,EO_PORT,ID,4,DINT_TO_STRING(ValoreScalato));END_IF;
					END_IF
			END_IF

	Status_Log:=1;
	Status_Vis:=16#2020F0;
END_IF
END_FUNCTION_BLOCK

(* POU Plant_Objects/obj_SW_CTB, ST *)
FUNCTION_BLOCK obj_SW_CTB
(* === Software Energy contabilizer [TICK=500ms] ===
   v1.0[16/04/05] - Versioning
*)
VAR_INPUT
	(* Settings *)
	ID				: BYTE;
	(* Physical Inputs *)
	T_SEND			: INT;  (* E-1 °C    *)
	T_RET			: INT;  (* E-1 °C    *)
	FLOW			: DINT; (* E-3 m^3/h *)
END_VAR
VAR_IN_OUT
	(* Persistent counter *)
	ENERGY_WH		: REAL;  (* Wh       *)
	ENERGY			: DWORD; (* E-2 MWh  *)
END_VAR
VAR_OUTPUT
	T_SEND_MEAN		: AVERAGE_INT;
	T_RET_MEAN		: AVERAGE_INT;
	FLOW_MEAN		: AVERAGE_DINT;
	POWER_KW		: REAL;
	(* Visu/Log *)
	Status_Log		: BYTE;
	Status_Vis		: DWORD;
END_VAR
VAR
	init			: BOOL;
	overflow		: BOOL;
	P_OLD			: REAL;

	(* HighSpeedLog *)
	hLog  : BOOL   :=FALSE;
	hFile : DWORD  :=0;
	hs1   : STRING;

END_VAR
(* Pv0[kW] = (FLOW/1000) * (8,164 *10 ^ -1 * T_SEND/10 + 9,623*10^2) * 4,186 * (T_SEND - T_RET)/10 / 3600 *)
(*POWER_KW := ( INT_TO_REAL(FLOW) * ( (8.164E-2 * INT_TO_REAL(T_SEND)) + 9.623E2 ) * 4.1868 * (T_SEND-T_RET) ) / 36000 ;*)

(* Pv1[kW] = ( FLOW * (-2.5987E-5 * T_SEND^2 - 1.8693E-2 * T_SEND + 1.0035E3) * 4.1868 * (T_SEND-T_RET) ) / 36E6 *)
POWER_KW := ( DINT_TO_REAL(FLOW) * ( (-2.5987E-5 * EXPT(T_SEND,2)) - (1.8693E-2 * T_SEND) + 1.0035E3 ) * 4.1868 * (T_SEND-T_RET) ) / 36E6 ;

(* Pv2[kW] = ( FLOW * (-2.19E-5 * T_SEND^2 - 2.81E-2 * T_SEND + 1.01E3) * 4.1868 * (T_SEND-T_RET) ) / 36E6 *)
(* ... *)

IF NOT init THEN
	init:=TRUE;
ELSE
	IF (POWER_KW + P_OLD)>0 THEN
		(* E[Wh] = ( (P0+P1)/2 ) * 0,5 / 3600 = (P0+P1)/14400 *)
		ENERGY_WH := ENERGY_WH + (( POWER_KW + P_OLD ) / 14.4);
	END_IF
END_IF

P_OLD:=POWER_KW;

IF ENERGY_WH>10000 THEN
	ENERGY_WH := ENERGY_WH - 10000;
	ENERGY := ENERGY + 1;
END_IF

(* Average of input values *)
T_SEND_MEAN(IN:=T_SEND);
T_RET_MEAN(IN:=T_RET);
FLOW_MEAN(IN:=FLOW);

(* Check status *)
Status_Log:=0; Status_Vis:=16#20F020;

hDbgLog();
END_FUNCTION_BLOCK
ACTION AddLogData:
Logger.s1:=INSERT('&CTB=',BYTE_TO_STRING(ID),4);
IF ID<10 THEN Logger.s1:=INSERT(Logger.s1,'0',4); END_IF
Mean();
Logger.s1:=CONCAT(Logger.s1,INT_TO_STRING(T_SEND_MEAN.AVG)					); Logger.s1:=CONCAT(Logger.s1,';');
Logger.s1:=CONCAT(Logger.s1,INT_TO_STRING(T_RET_MEAN.AVG)					); Logger.s1:=CONCAT(Logger.s1,';');
Logger.s1:=CONCAT(Logger.s1,DINT_TO_STRING(FLOW_MEAN.AVG)					); Logger.s1:=CONCAT(Logger.s1,';');
Mean_Reset();
Logger.s1:=CONCAT(Logger.s1,DINT_TO_STRING(REAL_TO_DINT(POWER_KW*1000))		); Logger.s1:=CONCAT(Logger.s1,';');
Logger.s1:=CONCAT(Logger.s1,DWORD_TO_STRING(ENERGY)							); Logger.s1:=CONCAT(Logger.s1,';');
Logger.s1:=CONCAT(Logger.s1,BYTE_TO_STRING(Status_Log)						);
ADDSTRING(ADR(Logger.TData), ADR(Logger.s1), Logger.TLen);
END_ACTION
ACTION hDbgLog:
IF hLog THEN
	IF hFile=0 THEN
		(* Open file *)
		hFile:=SysFileOpen('S:\HSLOG1.CSV','a');
		(* Start time *)
		hs1:=REPLACE( Sys.Time_LogString , ' ' , 1 , 11 );
		hs1:=CONCAT('>> Start', hs1);
		hs1:=CONCAT(hs1,Logger_CRLF);
		SysFileWrite(hFile, ADR(hs1), LEN(hs1));
		(* Data header *)
		hs1:='T-Send;T-Ret;Port;W;E';
		SysFileWrite(hFile, ADR(hs1), LEN(hs1));
	ELSE
		(* Log data *)
		hs1:=INT_TO_STRING(T_SEND);
		hs1:=CONCAT(hs1 , ';' );
		hs1:=CONCAT(hs1 , INT_TO_STRING(T_RET) );
		hs1:=CONCAT(hs1 , ';' );
		hs1:=CONCAT(hs1 , DINT_TO_STRING(FLOW) );
		hs1:=CONCAT(hs1 , ';' );
		hs1:=CONCAT(hs1 , REAL_TO_STRING(POWER_KW) );
		hs1:=CONCAT(hs1 , ';' );
		hs1:=CONCAT(hs1 , REAL_TO_STRING(ENERGY_WH) );
		hs1:=CONCAT(hs1 , Logger_CRLF );
		SysFileWrite(hFile, ADR(hs1), LEN(hs1));
	END_IF
ELSE
	IF hFile<>0 THEN
		(* Start time *)
		hs1:=REPLACE( Sys.Time_LogString , ' ' , 1 , 11 );
		hs1:=CONCAT('>> Stop', hs1);
		hs1:=CONCAT(hs1,Logger_CRLF);
		SysFileWrite(hFile, ADR(hs1), LEN(hs1));
		(* Close file *)
		SysFileClose(hFile);
		hFile:=0;
	END_IF
END_IF
END_ACTION
ACTION Mean:
T_SEND_MEAN.Read();
T_RET_MEAN.Read();
FLOW_MEAN.Read();
END_ACTION
ACTION Mean_Reset:
T_SEND_MEAN.Reset();
T_RET_MEAN.Reset();
FLOW_MEAN.Reset();
END_ACTION

(* POU Plant_Objects/obj_TPV, ST *)
FUNCTION_BLOCK obj_TPV
(* === TEMPERATURE PROBE  ===
   v1.0[16/04/15] - Versioning
*)
VAR CONSTANT
	NormalEv		: BYTE := 0;
	ErrorEv			: BYTE := 1;
	WarningEv		: BYTE := 2;
END_VAR
VAR_INPUT
	(* Settings *)
	ID				: BYTE;
	TAP				: BYTE:=4;	   (* Consecutive checks filter *)
	INITEV			: BOOL:= TRUE; (* Generate init OK event *)
	IN_EMIN			: INT :=-2000; (* Low error limit *)
	IN_WMIN			: INT := -550; (* Low warning value *)
	IN_WMAX			: INT :=  900; (* High warning value *)
	IN_EMAX			: INT := 8500; (* High error limit *)
	ERR_MIN_SHORT	: BOOL:= TRUE; (* TRUE  ==> EMIN=Short        , EMAX=Disconnected
									  FALSE ==> EMIN=Disconnected , EMAX=Short 		 *)
	(* Physical input *)
	IN			: INT;
END_VAR
VAR_OUTPUT
	WRN			: BOOL;	(* Value in warning range *)
	ERR			: BOOL;	(* Value error *)
	HI			: INT;	(* Highest value - cleared by Stat_Reset() action *)
	AVG			: INT; 	(* Average value - updated by Mean() action, cleared by Mean_Reset() action *)
	LOW			: INT;	(* Lowest value  - cleared by Stat_Reset() action *)

	Status_Log	: WORD;
	Status_Vis	: DWORD;
END_VAR
VAR
	cnt			: BYTE;
	event		: BYTE := 0;	(* 0: monitoring a generic, 1: monitoring an error, 2: monitoring a warning *)
	asum		: DINT;
	acnt		: WORD;
END_VAR
(* Check probe value limits *)
IF IN<=IN_EMIN OR IN>=IN_EMAX THEN
	IF NOT ERR THEN
		IF event <> ErrorEv THEN
			cnt := 1;
			event := ErrorEv;
		ELSE
			cnt:=cnt+1;
		END_IF

		IF cnt>TAP THEN
			cnt:=0;
			ERR:=TRUE; WRN:=FALSE;
			IF ( ERR_MIN_SHORT=TRUE  AND IN<=IN_EMIN ) OR ( ERR_MIN_SHORT=FALSE AND IN>=IN_EMAX ) THEN
				LogEv(EL_Alarm,EO_TPV,ID,5,INT_TO_STRING(IN));
			ELSE
				LogEv(EL_Alarm,EO_TPV,ID,4,INT_TO_STRING(IN));
			END_IF
		END_IF
	END_IF
ELSIF IN<=IN_WMIN OR IN>=IN_WMAX THEN
	IF NOT WRN THEN
		IF event <> WarningEv THEN
			cnt := 1;
			event := WarningEv;
		ELSE
			cnt:=cnt+1;
		END_IF

		IF cnt>TAP THEN
			cnt:=0;
			ERR:=FALSE; WRN:=TRUE;
			LogEv(EL_Wrn,EO_TPV,ID,SEL(IN<=IN_WMIN,3,2),INT_TO_STRING(IN));
		END_IF
	END_IF
ELSE
	IF INITEV OR WRN OR ERR THEN
		IF event <> NormalEv THEN
			cnt := 1;
			event := NormalEv;
		ELSE
			cnt:=cnt+1;
		END_IF

		IF cnt>TAP THEN
			cnt:=0;
			INITEV:=FALSE; ERR:=FALSE; WRN:=FALSE;
			LogEv(EL_Log,EO_TPV,ID,1,'Probe_OK');
		END_IF
	END_IF
END_IF


(*
(* Average value *)
IF acnt>=500 THEN
	Mean();
	asum := asum - AVG;
	acnt := acnt - 1;
END_IF

asum := asum + IN;
acnt := acnt + 1;
*)

AVG := IN;



(* Statistics values *)
IF IN<LOW THEN LOW:=IN; END_IF
IF IN>HI  THEN HI :=IN; END_IF


(* Status Log *)
IF ERR THEN	Status_Log := 2; Status_Vis := COLOR_RED;
ELSIF WRN THEN Status_Log := 1;	Status_Vis := COLOR_YELLOW;
ELSE Status_Log := 0; Status_Vis := COLOR_GREEN;
END_IF
END_FUNCTION_BLOCK
ACTION AddLogData:
Logger.s1:=INSERT('&TPV=',BYTE_TO_STRING(ID),4);
IF ID<10 THEN Logger.s1:=INSERT(Logger.s1,'0',4); END_IF
(*
Mean();
*)
Logger.s1:=CONCAT(Logger.s1,INT_TO_STRING(AVG));		Logger.s1:=CONCAT(Logger.s1,';');

Logger.s1:=CONCAT(Logger.s1,WORD_TO_STRING(Status_Log));
ADDSTRING(ADR(Logger.TData), ADR(Logger.s1), Logger.TLen);
END_ACTION
ACTION Mean:
AVG := DINT_TO_INT(asum/acnt);
END_ACTION
ACTION Mean_Reset:
AVG:=IN;
asum:=IN;
acnt:=1;
END_ACTION
ACTION Stat_Reset:
HI:=IN;
LOW:=IN;
END_ACTION

(* POU Plant_Objects/obj_TPV2, ST *)
FUNCTION_BLOCK obj_TPV2
(* === TEMPERATURE PROBE  ===
   v1.0[16/04/05] - Versioning
   v1.1[17/04/05] - Create status and VALID flag
*)
VAR_INPUT
	(* Settings *)
	ID				: BYTE;
	TAP				: BYTE:=4;	   (* Consecutive checks filter *)
	INITEV			: BOOL:= TRUE; (* Generate init OK event *)
	IN_EMIN			: INT :=-2000; (* Low error limit *)
	IN_WMIN			: INT := -550; (* Low warning value *)
	IN_WMAX			: INT :=  900; (* High warning value *)
	IN_EMAX			: INT := 8500; (* High error limit *)
	ERR_MIN_SHORT	: BOOL:= TRUE; (* TRUE  ==> EMIN=Short        , EMAX=Disconnected
									  FALSE ==> EMIN=Disconnected , EMAX=Short 		 *)
	(* Physical input *)
	IN				: INT;
END_VAR
VAR_OUTPUT
	(* Value outputs *)
	OUT			: INT;
	OUT_VALID	: BOOL;
	HI			: INT;	(* Highest value - cleared by Stat_Reset() action *)
	AVG			: INT; 	(* Average value - updated by Mean() action, cleared by Mean_Reset() action *)
	LOW			: INT;	(* Lowest value  - cleared by Stat_Reset() action *)
	(* Status *)
	Status_Log	: BYTE;
	Status_Vis 	: DWORD;
END_VAR
VAR
	cnt			: BYTE;
	asum		: DINT;
	acnt		: WORD;
END_VAR
(* Check probe value limits *)
IF IN<=IN_EMIN OR IN>=IN_EMAX THEN
	IF Status_Log<>2 THEN
		cnt:=cnt+1;
		IF cnt>TAP THEN
			cnt:=0;
			OUT_VALID:=FALSE;
			Status_Log:=2; Status_Vis:=16#2020F0;
			IF ( ERR_MIN_SHORT=TRUE  AND IN<=IN_EMIN ) OR ( ERR_MIN_SHORT=FALSE AND IN>=IN_EMAX ) THEN
				LogEv(EL_Alarm,EO_TPV,ID,5,INT_TO_STRING(IN));
			ELSE
				LogEv(EL_Alarm,EO_TPV,ID,4,INT_TO_STRING(IN));
			END_IF
		END_IF
	END_IF
ELSIF IN<=IN_WMIN OR IN>=IN_WMAX THEN
	IF NOT WRN THEN
		cnt:=cnt+1;
		IF cnt>TAP THEN
			cnt:=0;
			ERR:=FALSE; WRN:=TRUE;
			LogEv(EL_Wrn,EO_TPV,ID,SEL(IN<=IN_WMIN,3,2),INT_TO_STRING(IN));
		END_IF
	END_IF
ELSE
	IF init OR Status_Log>0 THEN
		cnt:=cnt+1;
		IF cnt>TAP THEN
			cnt:=0;
			INITEV:=FALSE;
			OUT_VALID:=TRUE;
			LogEv(EL_Log,EO_TPV,ID,1,'Probe_OK');

		END_IF
	END_IF
END_IF

(* Calculate statistics on valid values *)
IF OUT_VALID THEN

	(* Average value *)
	IF acnt>=60000 THEN
		Mean();
		asum := asum - AVG;
		acnt := acnt - 1;
	END_IF
	
	asum := asum + IN;
	acnt := acnt + 1;
	
	(* Statistics values *)
	IF IN<LOW THEN LOW:=IN; END_IF
	IF IN>HI  THEN HI :=IN; END_IF

END_IF
END_FUNCTION_BLOCK
ACTION Mean:
AVG := DINT_TO_INT(asum/acnt);
END_ACTION
ACTION Mean_Reset:
AVG:=IN;
asum:=IN;
acnt:=1;
END_ACTION
ACTION Stat_Reset:
HI:=IN;
LOW:=IN;
END_ACTION

(* POU Plant_Objects/obj_TPV_SENS, ST *)
FUNCTION_BLOCK obj_TPV_SENS
(* === TEMPERATURE PROBE FROM ANALOG INPUT ===
   v1.0[16/04/05] - Versioning
*)
VAR_INPUT
	(* Settings *)
	ID				: BYTE;
	PuntoMinX		: INT;			(* Parametri per la scalatura *)
	PuntoMaxX		: INT;
	PuntoMinY		: REAL;
	PuntoMaxY		: REAL;
	Decimali		: BYTE:=1;
	SogliaHH		: WORD;			(* Soglia per segnalazione Allarme Extra Range in alto - Solitamente sondo in CC *)
	SogliaHL		: WORD;			(* Soglia per segnalazione Allarme Extra Range in Basso - Solitamente sondo Aperta *)
	SogliaWH		: REAL;			(* Soglia per segnalazione Warning  in alto  *)
	SogliaWL		: REAL;    		(* Soglia per segnalazione Warning in basso  *)
	TAP				: INT:=2000;	(* Filtro in msec *)
	INITEV			: BOOL:= TRUE;	(* Generate init OK event *)
	(* Physical input *)
	AI_INPUT		: WORD;    		(* Sensor analog input *)
END_VAR
VAR_OUTPUT
	WRN				: BOOL;	(* Segnalazione Warning *)
	ERR				: BOOL; (* Segnalazione Errore *)
	ValoreScalato	: INT;
	(* Status *)
	Status_Log	: BYTE;
	Status_Vis 	: DWORD;
END_VAR
VAR
	SegnaleHH	: BOOL;
	SegnaleHL	: BOOL;
	SegnaleOK	: BOOL;
	SegnaleWH	: BOOL;
	SegnaleWL	: BOOL;
    FiltroWRN	: TON;
    FiltroOK	: TON;
    FiltroERR	: TON;
END_VAR
(* Verifico che le variabile letta dall'ingresso Analogico  sia dentro i range
ATTENZIONE I LIMITI SPESSO SONO IN WORD VERIFICA  TABELLA MANUALE WAGO  *)

SegnaleHH:=(AI_INPUT>=SogliaHH);
SegnaleHL:=(AI_INPUT<=SogliaHL);
SegnaleOK:=NOT (SegnaleHH OR SegnaleHL);

(* Linerarizzo il segnale di ingresso e la converto in unita ingegneristiche *)
ValoreScalato:=LINEAR_BAD(PuntoMinX, PuntoMaxX, AI_INPUT, PuntoMinY, PuntoMaxY, Decimali);


IF SegnaleOK  THEN
	(*  Verifica  e segnalazione Warning *)
	SegnaleWH:=(ValoreScalato>SogliaWH*(EXPT(10, Decimali)));
	SegnaleWL:=(ValoreScalato<SogliaWL*(EXPT(10, Decimali)));

	Status_Log:=0;
	Status_Vis:=16#20F020;    (* Indicazione WEB Visu Sonda OK *)

	FiltroWRN( IN:=(SegnaleWH OR SegnaleWL), PT:=INT_TO_TIME(TAP) );    (* Filtro su LOG *)
	IF  FiltroWRN.Q THEN     (* Condizione di WARNING *)
		IF NOT WRN THEN
			WRN:=TRUE;
			Status_Log:=1;
			LogEv(EL_Wrn,EO_TPV,ID,SEL(ValoreScalato<=SogliaWL,3,2),INT_TO_STRING(ValoreScalato));
		END_IF
	END_IF

    IF (INITEV OR WRN OR ERR) AND NOT FiltroWRN.Q THEN
		FiltroWRN(IN:=FALSE  , PT:=INT_TO_TIME(TAP));    (* Resetto il Filtro su LOG WRN  *)
		FiltroERR(IN:=FALSE  , PT:=INT_TO_TIME(TAP));    (* Resetto il Filtro su LOG ERR *)
		INITEV:=FALSE; ERR:=FALSE; WRN:=FALSE;
		LogEv(EL_Log,EO_TPV,ID,1,'');
	END_IF
ELSE
	FiltroERR(IN:=TRUE  , PT:= INT_TO_TIME(TAP) );    (* Filtro su LOG *)
	IF  FiltroERR.Q THEN     (* Condizione di WARNING *)
		IF NOT ERR THEN
			ERR:=TRUE;
			Status_Log:=2;

			IF SegnaleHH THEN LogEv(EL_Alarm,EO_TPV,ID,6,INT_TO_STRING(ValoreScalato));END_IF;
			IF SegnaleHL THEN LogEv(EL_Alarm,EO_TPV,ID,4,INT_TO_STRING(ValoreScalato));END_IF;
		END_IF
	END_IF

	Status_Vis:=16#2020F0;   (* Indicazione WEB Visu Sonda KO *)
END_IF



(* Status Log *)
IF ERR THEN
	Status_Log := 2;
	Status_Vis := COLOR_RED;
ELSIF WRN THEN
	Status_Log := 1;
	Status_Vis := COLOR_YELLOW;
ELSE
	Status_Log := 0; Status_Vis := COLOR_GREEN;
END_IF
END_FUNCTION_BLOCK
ACTION AddLogData:
Logger.s1:=INSERT('&TPV=',BYTE_TO_STRING(ID),4);
IF ID<10 THEN Logger.s1:=INSERT(Logger.s1,'0',4); END_IF

Logger.s1:=CONCAT(Logger.s1,INT_TO_STRING(ValoreScalato));		Logger.s1:=CONCAT(Logger.s1,';');

Logger.s1:=CONCAT(Logger.s1,WORD_TO_STRING(Status_Log));
ADDSTRING(ADR(Logger.TData), ADR(Logger.s1), Logger.TLen);
END_ACTION

(* POU Plant_Objects/obj_TPV_SENS2, ST *)
FUNCTION_BLOCK obj_TPV_SENS2
(* === TEMPERATURE PROBE FROM ANALOG INPUT ===
   v2.0[17/04/05] - Versioning
*)
VAR_INPUT
	(* Settings *)
	ID				: BYTE;
	TAP				: BYTE:=4;	   (* Consecutive checks filter *)
	INITEV			: BOOL:= TRUE; (* Generate init OK event *)
	IN_EMIN			: INT :=-2000; (* Low error limit *)
	IN_WMIN			: INT := -550; (* Low warning value *)
	IN_WMAX			: INT :=  900; (* High warning value *)
	IN_EMAX			: INT := 8500; (* High error limit *)
	ERR_MIN_SHORT	: BOOL:= TRUE; (* TRUE  ==> EMIN=Short        , EMAX=Disconnected
									  FALSE ==> EMIN=Disconnected , EMAX=Short 		 *)
	SCALE_LO_IN		: WORD;
	SCALE_LO_OUT	: INT;
	SCALE_HI_IN		: WORD;
	SCALE_HI_OUT	: INT;

	(* Physical input *)
	IN				: WORD;			(* Sensor analog input *)

	(* Settings *)
	PuntoMinX		: INT;			(* Parametri per la scalatura *)
	PuntoMaxX		: INT;
	PuntoMinY		: REAL;
	PuntoMaxY		: REAL;

	SogliaHH		: WORD;			(* Soglia per segnalazione Allarme Extra Range in alto - Solitamente sondo in CC *)
	SogliaHL		: WORD;			(* Soglia per segnalazione Allarme Extra Range in Basso - Solitamente sondo Aperta *)
	SogliaWH		: REAL;			(* Soglia per segnalazione Warning  in alto  *)
	SogliaWL		: REAL;    		(* Soglia per segnalazione Warning in basso  *)
END_VAR
VAR_OUTPUT
	OUT			: INT;
	OUT_VALID	: BOOL;
	(* Status *)
	Status_Log	: BYTE;
	Status_Vis 	: DWORD;
END_VAR
VAR
	SegnaleHH	: BOOL;
	SegnaleHL	: BOOL;
	SegnaleOK	: BOOL;
	SegnaleWH	: BOOL;
	SegnaleWL	: BOOL;
    FiltroWRN	: TON;
    FiltroOK	: TON;
    FiltroERR	: TON;
END_VAR
(* Verifico che le variabile letta dall'ingresso Analogico  sia dentro i range
ATTENZIONE I LIMITI SPESSO SONO IN WORD VERIFICA  TABELLA MANUALE WAGO  *)

SegnaleHH:=(AI_INPUT>=SogliaHH);
SegnaleHL:=(AI_INPUT<=SogliaHL);
SegnaleOK:=NOT (SegnaleHH OR SegnaleHL);

(* Linerarizzo il segnale di ingresso e la converto in unita ingegneristiche *)
OUT:=LINEAR_BAD(PuntoMinX, PuntoMaxX, AI_INPUT, PuntoMinY, PuntoMaxY, Decimali);


IF SegnaleOK  THEN
	(*  Verifica  e segnalazione Warning *)
	SegnaleWH:=(OUT > SogliaWH*(EXPT(10, Decimali)));
	SegnaleWL:=(OUT < SogliaWL*(EXPT(10, Decimali)));

	FiltroWRN( IN:=(SegnaleWH OR SegnaleWL), PT:=INT_TO_TIME(TAP) );    (* Filtro su LOG *)
	IF  FiltroWRN.Q THEN     (* Condizione di WARNING *)
		IF NOT WRN THEN
			WRN:=TRUE;
			LogEv(EL_Wrn,EO_TPV,ID,SEL(ValoreScalato<=SogliaWL,3,2),INT_TO_STRING(ValoreScalato));
		END_IF
	END_IF

    IF (INITEV OR WRN OR ERR) AND NOT FiltroWRN.Q THEN
		FiltroWRN(IN:=FALSE  , PT:=INT_TO_TIME(TAP));    (* Resetto il Filtro su LOG WRN  *)
		FiltroERR(IN:=FALSE  , PT:=INT_TO_TIME(TAP));    (* Resetto il Filtro su LOG ERR *)
		INITEV:=FALSE; ERR:=FALSE; WRN:=FALSE;
		LogEv(EL_Log,EO_TPV,ID,1,'');
	END_IF

	Status_Vis:=16#20F020;    (* Indicazione WEB Visu Sonda OK *)
ELSE
	FiltroERR(IN:=TRUE  , PT:= INT_TO_TIME(TAP) );    (* Filtro su LOG *)
	IF  FiltroERR.Q THEN     (* Condizione di WARNING *)
		IF NOT ERR THEN
			ERR:=TRUE;
			IF SegnaleHH THEN LogEv(EL_Alarm,EO_TPV,ID,6,INT_TO_STRING(ValoreScalato));END_IF;
			IF SegnaleHL THEN LogEv(EL_Alarm,EO_TPV,ID,4,INT_TO_STRING(ValoreScalato));END_IF;
		END_IF
	END_IF

	Status_Vis:=16#2020F0;   (* Indicazione WEB Visu Sonda KO *)
END_IF
END_FUNCTION_BLOCK

(* POU PLC_WDT, ST *)
FUNCTION PLC_WDT: DWORD VAR_INPUT dwEvent: DWORD; dwFilter: DWORD; dwOwner: DWORD; END_VAR
LogEv(EL_AlarmStop,EO_SYS,1,10,'Watchdog');
END_FUNCTION

(* POU Utils Functions/RAW16TOHEXSTR, ST *)
FUNCTION RAW16TOHEXSTR : STRING(128)
VAR_INPUT
	pData: POINTER TO BYTE;
	DataLen: BYTE;
END_VAR
VAR
	pt: POINTER TO BYTE;
	xl: BYTE;
END_VAR
pt:=ADR(RAW16TOHEXSTR);
xl:=0;

WHILE DataLen>0 AND xl<120 DO

	pData:=pData+1;

	pt^ := (pData^ / 16#10) + 48 + (((pData^ / 16#10)/10)*7);
	pt:=pt+1;
	pt^ := (pData^ AND 16#0F)  + 48 + (((pData^ AND 16#0F)/10)*7);
	pt:=pt+1;

	pData:=pData-1;

	pt^ := (pData^ / 16#10) + 48 + (((pData^ / 16#10)/10)*7);
	pt:=pt+1;
	pt^ := (pData^ AND 16#0F)  + 48 + (((pData^ AND 16#0F)/10)*7);
	pt:=pt+1;

	xl:=xl+4;

	DataLen:=DataLen-2;
	pData:=pData+2;

END_WHILE

pt^:=0;
END_FUNCTION

(* POU Utils Functions/RAWTOHEXSTR, ST *)
FUNCTION RAWTOHEXSTR : STRING(128)
VAR_INPUT
	pData: POINTER TO BYTE;
	DataLen: BYTE;
END_VAR
VAR
	pt: POINTER TO BYTE;
	xl: BYTE;
END_VAR
pt:=ADR(RAWTOHEXSTR);

xl:=2;

WHILE DataLen>0 AND xl<128 DO

	pt^ := (pData^ / 16#10) + 48 + (((pData^ / 16#10)/10)*7);
	pt:=pt+1;
	pt^ := (pData^ AND 16#0F)  + 48 + (((pData^ AND 16#0F)/10)*7);
	pt:=pt+1;

	xl:=xl+2;

	DataLen:=DataLen-1;
	pData:=pData+1;

END_WHILE

pt^:=0;
END_FUNCTION

(* POU Utils/RTC_Update, ST *)
FUNCTION RTC_Update : BOOL
VAR
	T: DT;
	TS: STRING;
	TS2: STRING;
	Hour: BYTE;
	Minute: BYTE;


END_VAR
(* Get RTC time *)
T:=SysRtcGetTime(TRUE);
Sys.Time_CT_DT:=T;
(* Calculate variables *)
TS:=DT_TO_STRING(T);
Sys.Time_LogString:=DELETE(STR:=TS, LEN:=3, POS:=1);
TS2:=MID(STR:=TS, LEN:=4, POS:= 4); Sys.Time_Year 	:=STRING_TO_WORD(TS2);
TS2:=MID(STR:=TS, LEN:=2, POS:= 9); Sys.Time_Month	:=STRING_TO_BYTE(TS2);
TS2:=MID(STR:=TS, LEN:=2, POS:=12); Sys.Time_Day  	:=STRING_TO_BYTE(TS2);
Sys.Time_CT_Day:=(32*(Sys.Time_Month-1)+Sys.Time_Day-1);
TS2:=MID(STR:=TS, LEN:=2, POS:=15); Hour			:=STRING_TO_BYTE(TS2);
TS2:=MID(STR:=TS, LEN:=2, POS:=18); Minute		 	:=STRING_TO_BYTE(TS2);
Sys.Time_CT_Quarter:=Hour*4+(Minute/15);


PrgDaylightSaving(xEnable:=TRUE , bWeekday=> NomeGiorno, xSummer=>OraLegale );
END_FUNCTION

